(* Logix 5000 project; controller AdvManLab vendor 1 type 14 code 158 rev 28.12; software revision 28.01; part 6 of 13 *)
(* tags used below, declared in another part *)
   Out : P_PF52x_Out;   // Common part of PF523 / PF525 Output Assembly
   Inp_FwdPermOK : BOOL;   // 1=Permissives OK, drive can start Forward
   Inp_FwdNBPermOK : BOOL;   // 1=Non-Bypassable Permissives OK, drive can start Forward
   Inp_RevPermOK : BOOL;   // 1=Permissives OK, drive can start Reverse
   Inp_RevNBPermOK : BOOL;   // 1=Non-Bypassable Permissives OK, motor can start Reverse
   Inp_IntlkOK : BOOL;   // 1=Interlocks OK, drive can start/run
   Inp_NBIntlkOK : BOOL;   // 1=Non-Bypassable Interlocks OK, drive can start/run
   Inp_OvrdCmd : SINT;   // Override Mode Command: 0=None, 1=Stop, 2=Start Fwd 3=Start Rev
   Cfg_SetTrack : BOOL;   // 1=PSets track OSets in Oper, OSets track PSets in Prog, 0=no tracking
   Cfg_PCmdClear : ALIAS FOR Mode.Cfg_PCmdClear;
   Cfg_ShedOnFailToStart : BOOL;   // 1=Stop Motor and Alarm on Fail to Start; 0=Alarm only on Fail to Start
   Cfg_ShedOnIOFault : BOOL;   // 1=Stop Motor and Alarm on I/O Fault; 0=Alarm only on I/O Fault
   Cfg_FailToStartAckReqd : ALIAS FOR FailToStart.Cfg_AckReqd;   // 1=Acknowledge required for Fail to Start Alarm
   Cfg_FailToStopAckReqd : ALIAS FOR FailToStop.Cfg_AckReqd;   // 1=Acknowledge required for Fail to Stop Alarm
   Cfg_IntlkTripAckReqd : ALIAS FOR IntlkTrip.Cfg_AckReqd;   // 1=Acknowledge required for Interlock Trip Alarm
   Cfg_DriveFaultAckReqd : ALIAS FOR DriveFault.Cfg_AckReqd;   // 1=Acknowledge required for Drive Fault Alarm
   Cfg_IOFaultAckReqd : ALIAS FOR IOFault.Cfg_AckReqd;   // 1=Acknowledge required for I/O Fault Alarm
   Cfg_FailToStartSeverity : ALIAS FOR FailToStart.Cfg_Severity;   // Fail To Start Alarm Severity: 1..250=Low, 251..500=Medium, 501..750=High, 751..1000=Urgent
   Cfg_FailToStopSeverity : ALIAS FOR FailToStop.Cfg_Severity;   // Fail To Stop Alarm Severity: 1..250=Low, 251..500=Medium, 501..750=High, 751..1000=Urgent
   Cfg_IntlkTripSeverity : ALIAS FOR IntlkTrip.Cfg_Severity;   // Interlock Trip Alarm Severity: 1..250=Low, 251..500=Medium, 501..750=High, 751..1000=Urgent
   Cfg_DriveFaultSeverity : ALIAS FOR DriveFault.Cfg_Severity;   // Drive Fault Alarm Severity: 1..250=Low, 251..500=Medium, 501..750=High, 751..1000=Urgent
   Cfg_IOFaultSeverity : ALIAS FOR IOFault.Cfg_Severity;   // I/O Fault Alarm Severity: 1..250=Low, 251..500=Medium, 501..750=High, 751..1000=Urgent
   Cfg_MaxSpdRef : REAL;   // Maximum Speed Reference in EU (for limiting)
   Cfg_SpeedRefRawMax : INT;   // Speed Reference Maximum in Drive (raw) Units (for scaling)
   Cfg_SpeedRefEUMax : REAL;   // Speed Reference Maximum in Engineering Units (for scaling)
   Cfg_SpeedFdbkRawMax : INT;   // Speed Feedback Maximum in Drive (raw) Units (for scaling)
   Cfg_SpeedFdbkEUMax : REAL;   // Speed Feedback Maximum in Engineering Units (for scaling)
   Cfg_SimRampT : DINT;   // Time to ramp speed fdbk when in Simulation (sec)
   Cfg_FailToStartT : DINT;   // Time after Start to get Run Feedback before Fault (sec)
   Cfg_FailToStopT : DINT;   // Time after Stop to drop Run Feedback before Fault (sec)
   Cfg_ResetPulseT : DINT;   // Time to pulse Out_Reset to clear drive fault
   PSet_Owner : DINT;   // Program Owner Request ID (non-zero) or Release (zero)
   PCmd_Start : BOOL;   // Program Command to Start Drive
   PCmd_Stop : BOOL;   // Program Command to Stop Drive
   PCmd_Fwd : BOOL;   // Program Command to set direction to Fowrard
   PCmd_Rev : BOOL;   // Program Command to set direction to Reverse
   PCmd_Reset : BOOL;   // Program Command to Reset drive fault and all Alarms requiring Reset
   OCmd_Start : BOOL;   // Operator Command to Start Drive
   OCmd_Stop : BOOL;   // Operator Command to Stop Drive
   OCmd_Jog : BOOL;   // Operator Command to Jog Drive (not cleared by P_PF52x!)
   OCmd_Fwd : BOOL;   // Operator Command to set direction to Forward
   OCmd_Rev : BOOL;   // Operator Command to set direction to Reverse
   OCmd_Bypass : BOOL;   // Operator Command to Bypass all Bypassable Interlocks and Permissives
   OCmd_Check : BOOL;   // Operator Command to Check (not bypass) all Interlocks and Permissives
   MCmd_Disable : BOOL;   // Maintenance Command to Disable Drive
   MCmd_Enable : BOOL;   // Maintenance Command to Enable (allow to run) Drive
   OCmd_Reset : BOOL;   // Operator Command to Reset all Alarms requiring Reset
   OCmd_ResetAckAll : BOOL;   // Operator Command to Reset all Alarms and latched Shed conditions
   Val_SpeedRefEUMax : REAL;   // Maximum of Speed Reference = MAX (Cfg_SpeedFdbkEUMin, Cfg_SpeedFdbkEUMax)
   Val_SpeedFdbkEUMax : REAL;   // Maximum of Speed Feedback = MAX (Cfg_SpeedFdbkEUMin, Cfg_SpeedFdbkEUMax)
   Val_OutPower : REAL;   // Drive output power (kW)
   Val_Cmd : SINT;   // Device Command 0=None, 1=Stop, 2=StartFwd 3=StartRev 4=JogFwd 5=JogRev
   Val_Fdbk : SINT;   // Device Feedback 0=Stopped, 1=Running Fwd 2=Running Rev 3=Accelerating 4=Decelerating
   Val_Sts : SINT;   // Device Confirmed Sts 0? 1=Stop 2=RunF 3=RunR 4=JogF 5=JogR 6=Stopping 7=Starting F 8=Starting R, 33=Disabled
   Val_Fault : SINT;   // Device Fault Status 0=None, 16=Fail to Start, 17 = Fail to Stop, 18=Drive Fault, 32=I/O Fault, 34=Config Error
   Val_Mode : ALIAS FOR Mode.Val;
   Val_Owner : DINT;   // Current Object Owner ID (0=not owned)
   Sts_ActualDir : BOOL;   // 1=Drive Actual direction is Forward, 0=Reverse
   Nrdy_OperPrio : BOOL;   // 1=Device Not Ready: Operator State 0 Priority Command Requires Reset
   Nrdy_Fail : BOOL;   // 1=Device Not Ready: Device Failure (Shed Requires Reset)
   Nrdy_IOFault : BOOL;   // 1=Device Not Ready: I/O Fault (Shed Requires Reset)
   Ack_FailToStart : ALIAS FOR FailToStart.Ack;   // 1=Fail to Start Alarm has been acknowledged
   Ack_FailToStop : ALIAS FOR FailToStop.Ack;   // 1=Fail to Stop Alarm has been acknowledged
   Ack_IntlkTrip : ALIAS FOR IntlkTrip.Ack;   // 1=Interlock Trip Alarm has been acknowledged
   Ack_DriveFault : ALIAS FOR DriveFault.Ack;   // 1=Drive Fault Alarm has been acknowledged
   Ack_IOFault : ALIAS FOR IOFault.Ack;   // 1=I/O Fault Alarm has been acknowledged
   P_PF52x : BOOL;   // Unique Parameter Name for auto - discovery
   Mode : P_Mode;   // Drive Mode Selection
   Wrk_Run : BOOL;   // 1=Drive should be "running", 0=should be "stopped"
   Wrk_Jog : BOOL;   // 1=Jog Drive, 0=Drive not jogging
(* P_PF52x, continued *)

ROUTINE Prescan   (* ladder *)
// Clear Ownership, set drive to STOP, clear "lurking" Commands
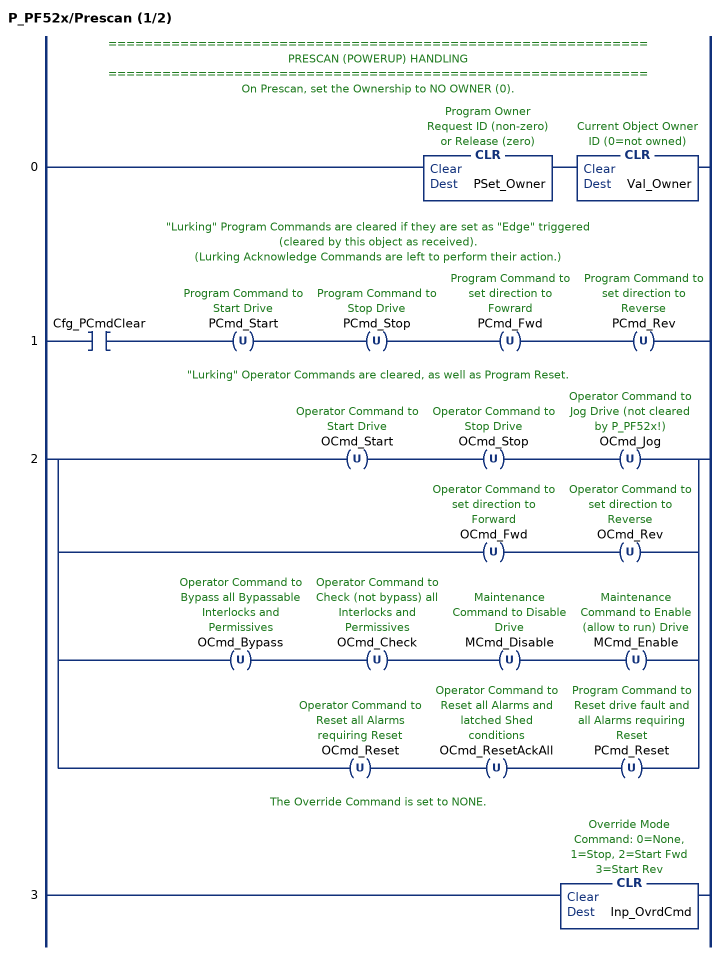
   // ============================================================
   // PRESCAN (POWERUP) HANDLING
   // ============================================================
   // On Prescan, set the Ownership to NO OWNER (0).
   0: CLR(PSet_Owner)CLR(Val_Owner);
   // "Lurking" Program Commands are cleared if they are set as "Edge" triggered
   // (cleared by this object as received).
   // (Lurking Acknowledge Commands are left to perform their action.)
   1: XIC(Cfg_PCmdClear)OTU(PCmd_Start)OTU(PCmd_Stop)OTU(PCmd_Fwd)OTU(PCmd_Rev);
   // "Lurking" Operator Commands are cleared, as well as Program Reset.
   2: [OTU(OCmd_Start) OTU(OCmd_Stop) OTU(OCmd_Jog) ,OTU(OCmd_Fwd) OTU(OCmd_Rev) ,OTU(OCmd_Bypass) OTU(OCmd_Check) OTU(MCmd_Disable) OTU(MCmd_Enable) ,OTU(OCmd_Reset) OTU(OCmd_ResetAckAll) OTU(PCmd_Reset) ];
   // The Override Command is set to NONE.
   3: CLR(Inp_OvrdCmd);
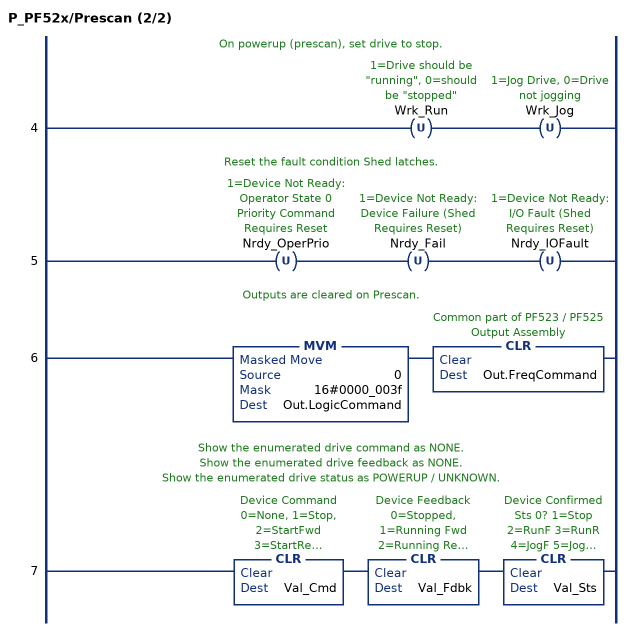
   // On powerup (prescan), set drive to stop.
   4: OTU(Wrk_Run)OTU(Wrk_Jog);
   // Reset the fault condition Shed latches.
   5: OTU(Nrdy_OperPrio)OTU(Nrdy_Fail)OTU(Nrdy_IOFault);
   // Outputs are cleared on Prescan.
   6: MVM(0,16#0000_003f,Out.LogicCommand)CLR(Out.FreqCommand);
   // Show the enumerated drive command as NONE.
   // Show the enumerated drive feedback as NONE.
   // Show the enumerated drive status as POWERUP / UNKNOWN.
   7: CLR(Val_Cmd)CLR(Val_Fdbk)CLR(Val_Sts);
END_ROUTINE
END_ADD_ON_INSTRUCTION

ADD_ON_INSTRUCTION PF525_Faceplate_AOI   (* revision 1.0 *)
// PF525 Drive FTView ME Faceplate AOI
VAR_INPUT
   Inp_NumRowsVis : DINT := 9;
   Set_FaceplateAnimation : INT;
END_VAR
VAR_OUTPUT
   Sts_ProgramModeEnabled : BOOL; {access Read Only}
   Sts_OperatorModeEnabled : BOOL; {access Read Only}
   Sts_DriveStatus_Faulted : BOOL; {access Read Only}
   Sts_DriveStatus_Active : BOOL; {access Read Only}
   Sts_DriveStatus_Ready : BOOL; {access Read Only}
   Sts_DriveStatus_Alarm : BOOL; {access Read Only}
   Sts_DriveStatus_AtSpeed : BOOL; {access Read Only}
   Sts_CommFault : BOOL; {access Read Only}
   Sts_DriveStatus_ActualDir : BOOL; {access Read Only}
   Sts_DeviceState : DINT; {access Read Only}
   Sts_Value1 : REAL; {access Read Only}
   Sts_Value2 : REAL; {access Read Only}
   Sts_Value3 : REAL; {access Read Only}
   Sts_Value4 : REAL; {access Read Only}
END_VAR
VAR_INPUT
   Set_TrendNextPenOper : DINT;
   Set_Value1Min : DINT;
   Set_Value1Max : DINT := 60;
   Set_Value2Min : DINT;
   Set_Value2Max : DINT := 1;
   Set_Value3Max : DINT := 1;
   Set_Value3Min : DINT;
END_VAR
VAR_OUTPUT
   Val_TrendMax : DINT; {access Read Only}
   Val_TrendMin : DINT; {access Read Only}
   Val_SpdFdbk_Units : DINT; {access Read Only}
   Val_Fault1Code : DINT; {access Read Only}
END_VAR
VAR_INPUT
   Cmd_OperOperReq : BOOL;
   Cmd_ProgOperReq : BOOL;
   Cmd_OperProgReq : BOOL;
   Cmd_ProgProgReq : BOOL;
   Cmd_StartOper : BOOL;
   Cmd_StartProg : BOOL;
   Cmd_StopOper : BOOL;
   Cmd_StopProg : BOOL;
   Cmd_ResetOper : BOOL;
   Cmd_ResetProg : BOOL;
   Cmd_JogOper : BOOL;
   Cmd_JogProg : BOOL;
   Cmd_FwdOper : BOOL;
   Cmd_FwdProg : BOOL;
   Cmd_RevOper : BOOL;
   Cmd_RevProg : BOOL;
   Cmd_OperToProgPermissive : BOOL := 1;
   Cmd_ProgToOperPermissive : BOOL := 1;
   Set_SpeedOper : INT;
END_VAR
VAR_IN_OUT
   Inp_PowerFlex_525 : AB:PowerFlex525V_E_8A02D441:I:0; {required}
   Out_PowerFlex_525 : AB:PowerFlex525V_E_5483BAFD:O:0; {required}
END_VAR
VAR_INPUT
   Cmd_MOPIncProg : BOOL;
   Cmd_MOPIncOper : BOOL;
   Cmd_Accel1Oper : BOOL;
   Cmd_Accel2Oper : BOOL;
   Cmd_Decel1Oper : BOOL;
   Cmd_Decel2Oper : BOOL;
   Cmd_Accel1Prog : BOOL;
   Cmd_Accel2Prog : BOOL;
   Cmd_Decel1Prog : BOOL;
   Cmd_Decel2Prog : BOOL;
   Cmd_MOPDecProg : BOOL;
   Cmd_MOPDecOper : BOOL;
   Set_AccelProg : REAL;
   Set_DecelProg : REAL;
   Set_CommFaultTimerPresetProg : DINT := 10000;
   Cmd_LocalContrlProg : BOOL;
   Cmd_LocalContrlOper : BOOL;
   Cmd_FreqSel01Prog : BOOL;
   Cmd_FreqSel01Oper : BOOL;
   Cmd_FreqSel02Prog : BOOL;
   Cmd_FreqSel02Oper : BOOL;
   Cmd_FreqSel03Prog : BOOL;
   Cmd_FreqSel03Oper : BOOL;
   Set_SpeedProg : INT;
   Set_CommFaultTimerPresetOper : DINT;
   Set_DecelOper : REAL;
   Set_AccelOper : REAL;
   Inp_FaultCode : DINT;   // Fault Code
   NotReady_Fault : BOOL;
   CLEAR_Fault : BOOL;
   Module_FaultTrigger : BOOL;
   Module_FaultCode : DINT;
   RESET_Fault : BOOL;
   Inp_Display_Val_1 : REAL;
   Inp_Display_Val_2 : REAL;
   Inp_Display_Val_3 : REAL;
   Inp_Display_Val_4 : REAL;
   Comm_Status : DINT;
   Sts_DriveStatus_CommFault : BOOL;
   Inst_Error : BOOL;
END_VAR
VAR_IN_OUT
   LastFault_Msg : MESSAGE; {required}
END_VAR
VAR_INPUT
   LastFaultCode : DINT;
   SpdRef_Units : INT;
   SpdScaler60Hz : REAL; {required}
   GearRatio : REAL; {required}
   Out_SpdRef_Units : DINT;
   Val_OutputFreq : REAL;
   Val_OutputCurrent : REAL;
   Val_OutputVoltage : DINT;
END_VAR
VAR_OUTPUT
   Sts_PowerflexAlarmTrigger : DINT; {access Read Only}
   Controller_trigger : BOOL; {access Read Only}
END_VAR
VAR
   Set_Value4Units : STRING := 'units';
   Set_Value3Units : STRING := 'units';
   Set_Value2Units : STRING := 'Amps';
   Set_Value1Units : STRING := 'Hz';
   Set_SpeedUnitsOper : STRING := 'Hz';
   Set_DeviceNameOper : STRING := 'PF525';
   Set_Value3Name : STRING := 'Value 3';
   Set_Value2Name : STRING := 'curr fdbk';
   Set_Value1Name : STRING := 'unit fdbk';
   Set_Value4Name : STRING := 'Value 4';
   OperONS : BOOL; {access None}
   CommFaultTimer : TIMER := (PRE := 10000); {access None}
   Trigger_ONS : BOOL;
   Trigger_Delay_Timer : TIMER; {access None}
   Handshake_Initial_Status : BOOL;
   Comm_Loss_Delay_Timer : TIMER; {access None}
   storage_bit2 : BOOL; {access None}
END_VAR

ROUTINE Logic   (* ladder *)
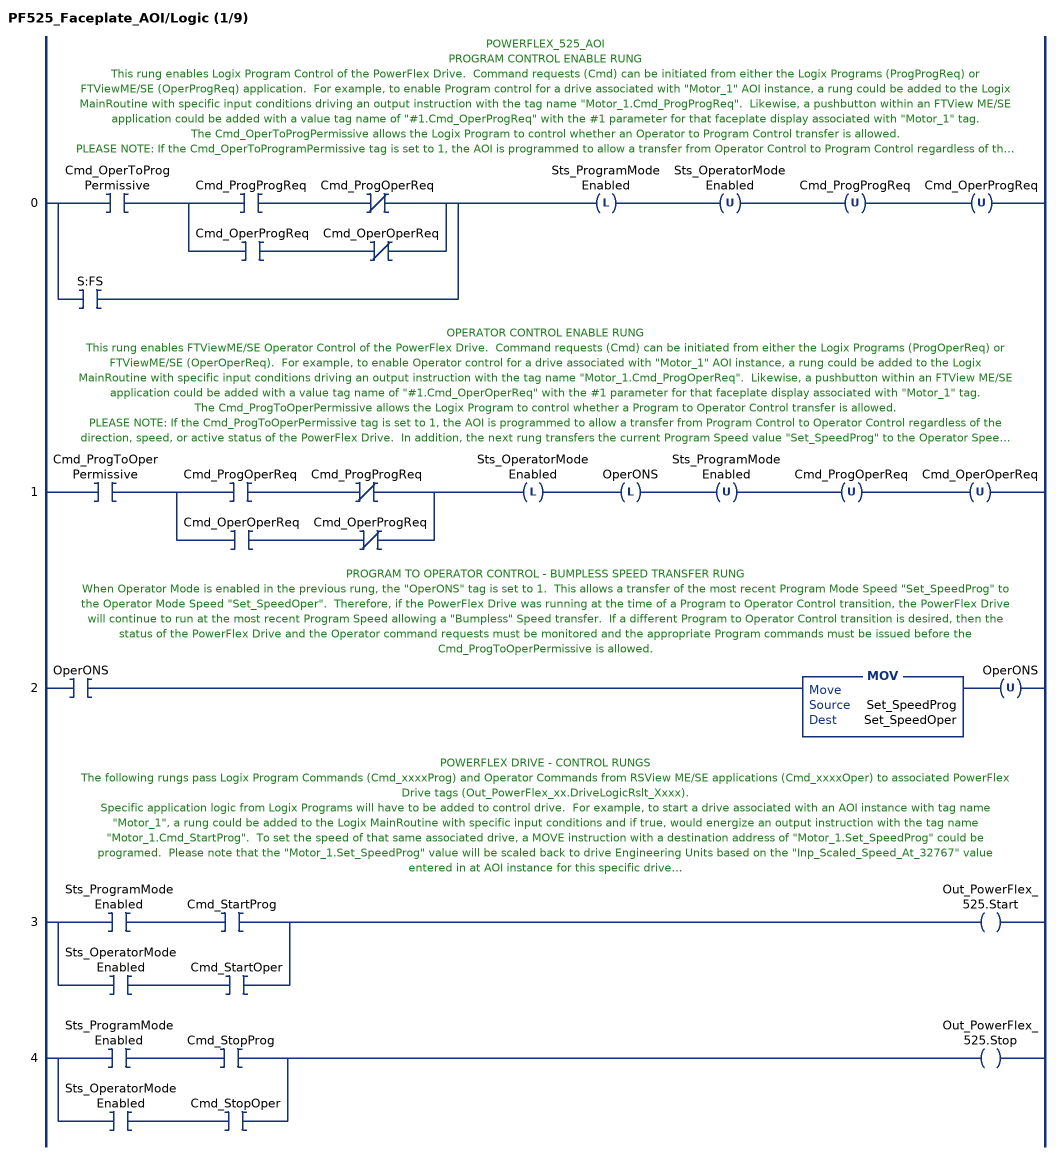
   // POWERFLEX_525_AOI
   // PROGRAM CONTROL ENABLE RUNG
   // This rung enables Logix Program Control of the PowerFlex Drive.  Command requests (Cmd) can be initiated from either the Logix Programs (ProgProgReq) or FTViewME/SE (OperProgReq) application.  For example, to enable Program control for a drive associated with "Motor_1" AOI instance, a rung could be added to the Logix MainRoutine with specific input conditions driving an output instruction with the tag name "Motor_1.Cmd_ProgProgReq".  Likewise, a pushbutton within an FTView ME/SE application could be added with a value tag name of "#1.Cmd_OperProgReq" with the #1 parameter for that faceplate display associated with "Motor_1" tag.
   // The Cmd_OperToProgPermissive allows the Logix Program to control whether an Operator to Program Control transfer is allowed.
   // PLEASE NOTE: If the Cmd_OperToProgramPermissive tag is set to 1, the AOI is programmed to allow a transfer from Operator Control to Program Control regardless of the direction, speed, or active status of the PowerFlex Drive.  Therefore, the status of the PowerFlex Drive must be monitored and used to set Cmd_OperToProgramPermissive tag outside of the AOI to insure a safe transfer.
   0: [XIC(Cmd_OperToProgPermissive) [XIC(Cmd_ProgProgReq) XIO(Cmd_ProgOperReq) ,XIC(Cmd_OperProgReq) XIO(Cmd_OperOperReq) ] ,XIC(S:FS) ]OTL(Sts_ProgramModeEnabled)OTU(Sts_OperatorModeEnabled)OTU(Cmd_ProgProgReq)OTU(Cmd_OperProgReq);
   // OPERATOR CONTROL ENABLE RUNG
   // This rung enables FTViewME/SE Operator Control of the PowerFlex Drive.  Command requests (Cmd) can be initiated from either the Logix Programs (ProgOperReq) or FTViewME/SE (OperOperReq).  For example, to enable Operator control for a drive associated with "Motor_1" AOI instance, a rung could be added to the Logix MainRoutine with specific input conditions driving an output instruction with the tag name "Motor_1.Cmd_ProgOperReq".  Likewise, a pushbutton within an FTView ME/SE application could be added with a value tag name of "#1.Cmd_OperOperReq" with the #1 parameter for that faceplate display associated with "Motor_1" tag.
   // The Cmd_ProgToOperPermissive allows the Logix Program to control whether a Program to Operator Control transfer is allowed.
   // PLEASE NOTE: If the Cmd_ProgToOperPermissive tag is set to 1, the AOI is programmed to allow a transfer from Program Control to Operator Control regardless of the direction, speed, or active status of the PowerFlex Drive.  In addition, the next rung transfers the current Program Speed value "Set_SpeedProg" to the Operator Speed tag, "Set_SpeedOper" tag, creating a "bumpless" transfer when a transfer from Program Control to Operator Control is executed.  Therefore, the status of the PowerFlex Drive must be monitored and appropriate Program commands, for the specific application, must be issued before the Cmd_ProgToOperPermissive tag is set, to insure a safe Program to Operator Control transfer.
   1: XIC(Cmd_ProgToOperPermissive)[XIC(Cmd_ProgOperReq) XIO(Cmd_ProgProgReq) ,XIC(Cmd_OperOperReq) XIO(Cmd_OperProgReq) ]OTL(Sts_OperatorModeEnabled)OTL(OperONS)OTU(Sts_ProgramModeEnabled)OTU(Cmd_ProgOperReq)OTU(Cmd_OperOperReq);
   // PROGRAM TO OPERATOR CONTROL - BUMPLESS SPEED TRANSFER RUNG
   // When Operator Mode is enabled in the previous rung, the "OperONS" tag is set to 1.  This allows a transfer of the most recent Program Mode Speed "Set_SpeedProg" to the Operator Mode Speed "Set_SpeedOper".  Therefore, if the PowerFlex Drive was running at the time of a Program to Operator Control transition, the PowerFlex Drive will continue to run at the most recent Program Speed allowing a "Bumpless" Speed transfer.  If a different Program to Operator Control transition is desired, then the status of the PowerFlex Drive and the Operator command requests must be monitored and the appropriate Program commands must be issued before the Cmd_ProgToOperPermissive is allowed.
   2: XIC(OperONS)MOV(Set_SpeedProg,Set_SpeedOper)OTU(OperONS);
   // POWERFLEX DRIVE - CONTROL RUNGS
   // The following rungs pass Logix Program Commands (Cmd_xxxxProg) and Operator Commands from RSView ME/SE applications (Cmd_xxxxOper) to associated PowerFlex Drive tags (Out_PowerFlex_xx.DriveLogicRslt_Xxxx).
   // Specific application logic from Logix Programs will have to be added to control drive.  For example, to start a drive associated with an AOI instance with tag name "Motor_1", a rung could be added to the Logix MainRoutine with specific input conditions and if true, would energize an output instruction with the tag name "Motor_1.Cmd_StartProg".  To set the speed of that same associated drive, a MOVE instruction with a destination address of "Motor_1.Set_SpeedProg" could be programed.  Please note that the "Motor_1.Set_SpeedProg" value will be scaled back to drive Engineering Units based on the "Inp_Scaled_Speed_At_32767" value entered in at AOI instance for this specific drive.
   // Commands from FTView ME/SE applications will also control the drive when Operator Mode is enabled.  For example, to start a drive associated with "Motor_1" AOI instance, a pushbutton within an FTView ME application with a tag name of "#1.Cmd_StartOper" would have to be configured.  The #1 parameter tagname for that faceplate display would have to be "Motor_1".  To set the speed of that same "Motor_1" associated drive, a numeric input object with the tag name of "#1.Set_SpeedOper" would have to be configured.  Please note that the "#1.Set_SpeedOper" value will be scaled back to drive Engineering Units based on the "Inp_Scaled_Speed_At_32767" value entered in at AOI instance for this specific drive.
   // For ability to set AccelTime1 and DecelTime1, the datalinks within the PowerFlex Drive Module Definitions need to be assigned to these drive parameters.
   3: [XIC(Sts_ProgramModeEnabled) XIC(Cmd_StartProg) ,XIC(Sts_OperatorModeEnabled) XIC(Cmd_StartOper) ]OTE(Out_PowerFlex_525.Start);
   4: [XIC(Sts_ProgramModeEnabled) XIC(Cmd_StopProg) ,XIC(Sts_OperatorModeEnabled) XIC(Cmd_StopOper) ]OTE(Out_PowerFlex_525.Stop);
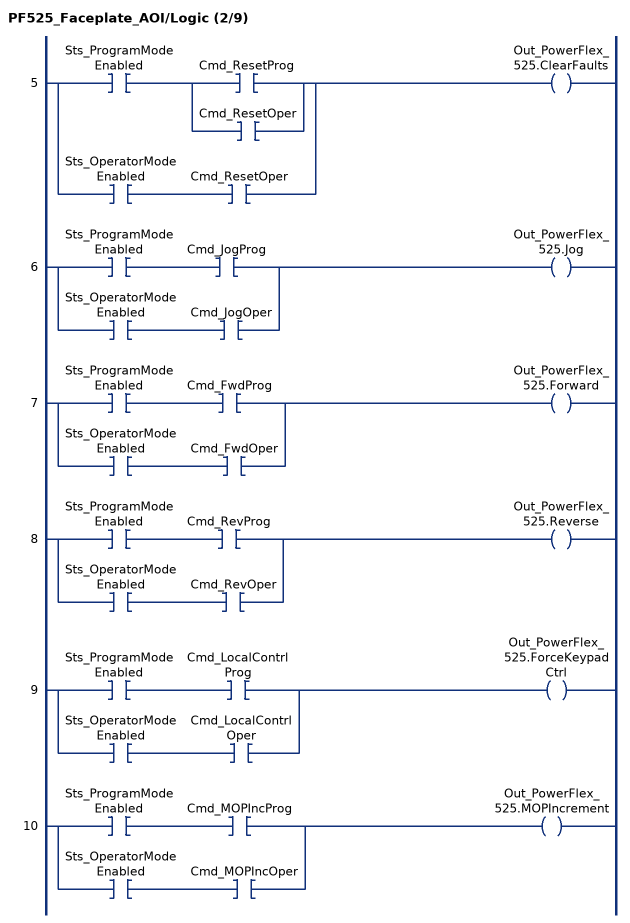
   5: [XIC(Sts_ProgramModeEnabled) [XIC(Cmd_ResetProg) ,XIC(Cmd_ResetOper) ] ,XIC(Sts_OperatorModeEnabled) XIC(Cmd_ResetOper) ]OTE(Out_PowerFlex_525.ClearFaults);
   6: [XIC(Sts_ProgramModeEnabled) XIC(Cmd_JogProg) ,XIC(Sts_OperatorModeEnabled) XIC(Cmd_JogOper) ]OTE(Out_PowerFlex_525.Jog);
   7: [XIC(Sts_ProgramModeEnabled) XIC(Cmd_FwdProg) ,XIC(Sts_OperatorModeEnabled) XIC(Cmd_FwdOper) ]OTE(Out_PowerFlex_525.Forward);
   8: [XIC(Sts_ProgramModeEnabled) XIC(Cmd_RevProg) ,XIC(Sts_OperatorModeEnabled) XIC(Cmd_RevOper) ]OTE(Out_PowerFlex_525.Reverse);
   9: [XIC(Sts_ProgramModeEnabled) XIC(Cmd_LocalContrlProg) ,XIC(Sts_OperatorModeEnabled) XIC(Cmd_LocalContrlOper) ]OTE(Out_PowerFlex_525.ForceKeypadCtrl);
   10: [XIC(Sts_ProgramModeEnabled) XIC(Cmd_MOPIncProg) ,XIC(Sts_OperatorModeEnabled) XIC(Cmd_MOPIncOper) ]OTE(Out_PowerFlex_525.MOPIncrement);
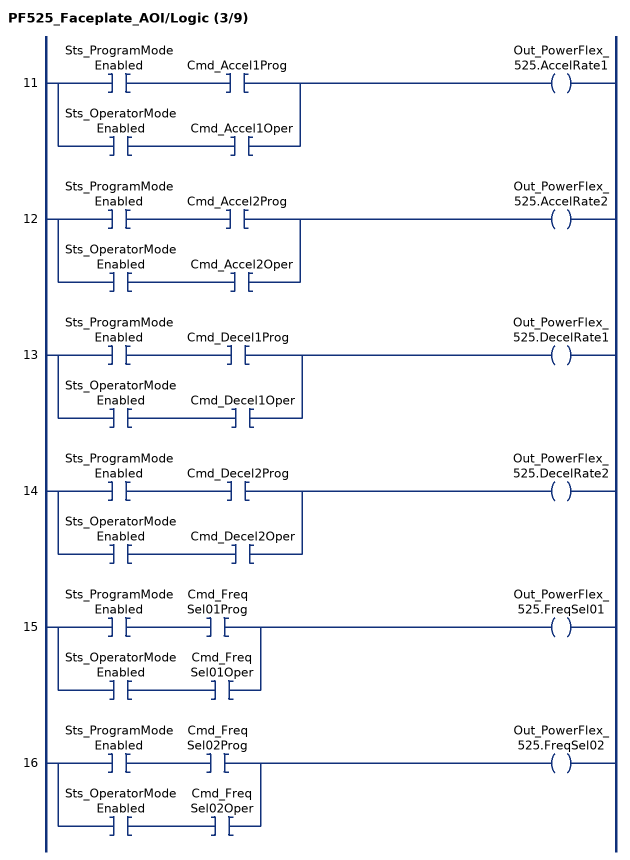
   11: [XIC(Sts_ProgramModeEnabled) XIC(Cmd_Accel1Prog) ,XIC(Sts_OperatorModeEnabled) XIC(Cmd_Accel1Oper) ]OTE(Out_PowerFlex_525.AccelRate1);
   12: [XIC(Sts_ProgramModeEnabled) XIC(Cmd_Accel2Prog) ,XIC(Sts_OperatorModeEnabled) XIC(Cmd_Accel2Oper) ]OTE(Out_PowerFlex_525.AccelRate2);
   13: [XIC(Sts_ProgramModeEnabled) XIC(Cmd_Decel1Prog) ,XIC(Sts_OperatorModeEnabled) XIC(Cmd_Decel1Oper) ]OTE(Out_PowerFlex_525.DecelRate1);
   14: [XIC(Sts_ProgramModeEnabled) XIC(Cmd_Decel2Prog) ,XIC(Sts_OperatorModeEnabled) XIC(Cmd_Decel2Oper) ]OTE(Out_PowerFlex_525.DecelRate2);
   15: [XIC(Sts_ProgramModeEnabled) XIC(Cmd_FreqSel01Prog) ,XIC(Sts_OperatorModeEnabled) XIC(Cmd_FreqSel01Oper) ]OTE(Out_PowerFlex_525.FreqSel01);
   16: [XIC(Sts_ProgramModeEnabled) XIC(Cmd_FreqSel02Prog) ,XIC(Sts_OperatorModeEnabled) XIC(Cmd_FreqSel02Oper) ]OTE(Out_PowerFlex_525.FreqSel02);
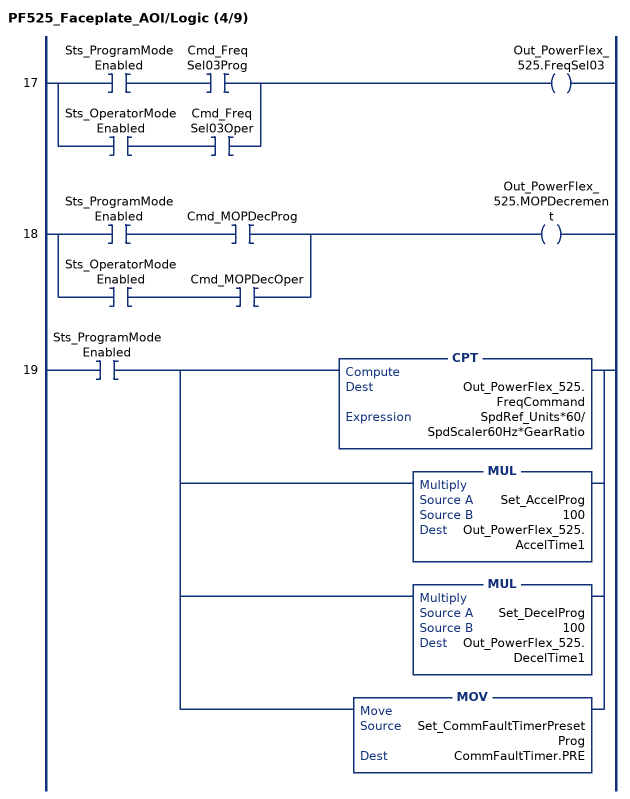
   17: [XIC(Sts_ProgramModeEnabled) XIC(Cmd_FreqSel03Prog) ,XIC(Sts_OperatorModeEnabled) XIC(Cmd_FreqSel03Oper) ]OTE(Out_PowerFlex_525.FreqSel03);
   18: [XIC(Sts_ProgramModeEnabled) XIC(Cmd_MOPDecProg) ,XIC(Sts_OperatorModeEnabled) XIC(Cmd_MOPDecOper) ]OTE(Out_PowerFlex_525.MOPDecrement);
   19: XIC(Sts_ProgramModeEnabled)[CPT(Out_PowerFlex_525.FreqCommand,SpdRef_Units*60/SpdScaler60Hz*GearRatio) ,MUL(Set_AccelProg,100,Out_PowerFlex_525.AccelTime1) ,MUL(Set_DecelProg,100,Out_PowerFlex_525.DecelTime1) ,MOV(Set_CommFaultTimerPresetProg,CommFaultTimer.PRE) ];
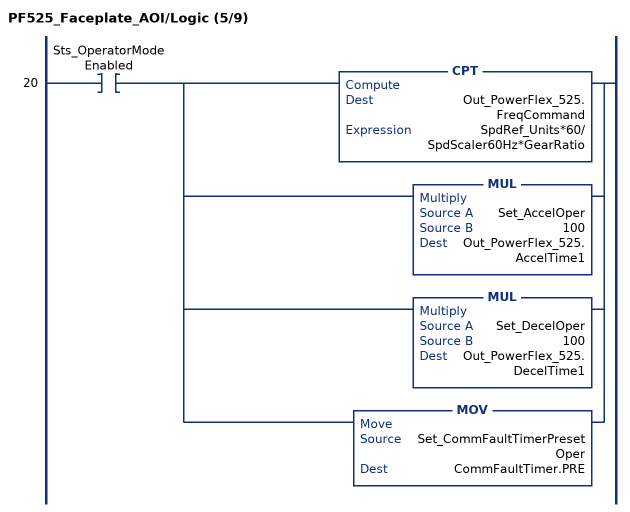
   20: XIC(Sts_OperatorModeEnabled)[CPT(Out_PowerFlex_525.FreqCommand,SpdRef_Units*60/SpdScaler60Hz*GearRatio) ,MUL(Set_AccelOper,100,Out_PowerFlex_525.AccelTime1) ,MUL(Set_DecelOper,100,Out_PowerFlex_525.DecelTime1) ,MOV(Set_CommFaultTimerPresetOper,CommFaultTimer.PRE) ];
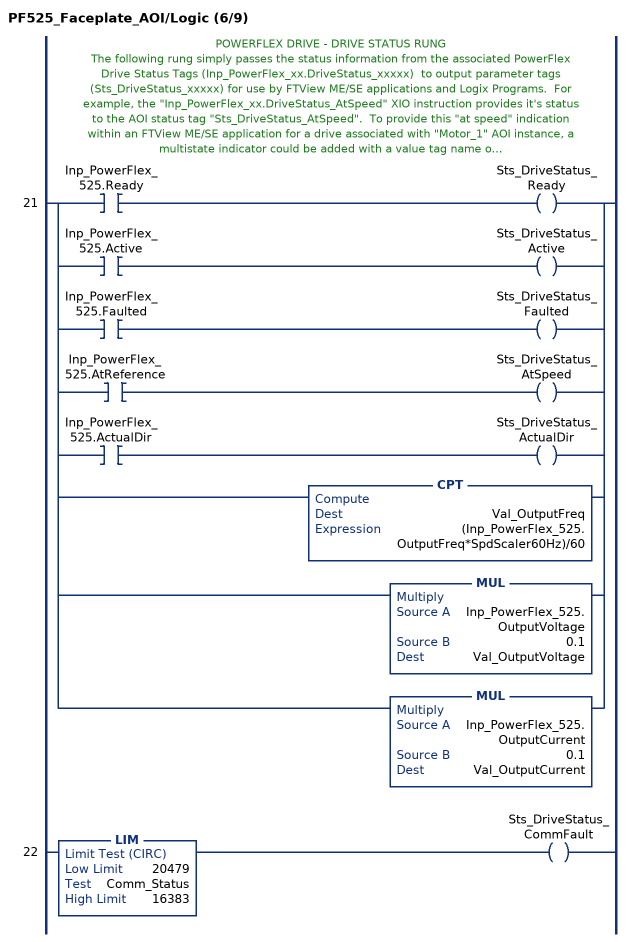
   // POWERFLEX DRIVE - DRIVE STATUS RUNG
   // The following rung simply passes the status information from the associated PowerFlex Drive Status Tags (Inp_PowerFlex_xx.DriveStatus_xxxxx)  to output parameter tags (Sts_DriveStatus_xxxxx) for use by FTView ME/SE applications and Logix Programs.  For example, the "Inp_PowerFlex_xx.DriveStatus_AtSpeed" XIO instruction provides it's status to the AOI status tag "Sts_DriveStatus_AtSpeed".  To provide this "at speed" indication within an FTView ME/SE application for a drive associated with "Motor_1" AOI instance, a multistate indicator could be added with a value tag name of "#1.Sts_DriveStatus_AtSpeed".  The #1 parameter for the faceplate display with the at speed indicator associated with "Motor_1" would be assigned the "Motor_1" tag.  To use this "Sts_DriveStatus_AtSpeed" status for the drive associated with "Motor_1" within a Logix Program routine you would simply assign an input instruction with a tag name of Motor_1.Sts_ DriveStatus_AtSpeed.  Please note that the "Val_OutputFreq" value used by the FTView ME/SE application is scaled based on the "Inp_Scaled_Speed_At_60Hz" value entered in at AOI instance for the specific drive.
   21: [XIC(Inp_PowerFlex_525.Ready) OTE(Sts_DriveStatus_Ready) ,XIC(Inp_PowerFlex_525.Active) OTE(Sts_DriveStatus_Active) ,XIC(Inp_PowerFlex_525.Faulted) OTE(Sts_DriveStatus_Faulted) ,XIC(Inp_PowerFlex_525.AtReference) OTE(Sts_DriveStatus_AtSpeed) ,XIC(Inp_PowerFlex_525.ActualDir) OTE(Sts_DriveStatus_ActualDir) ,CPT(Val_OutputFreq,(Inp_PowerFlex_525.OutputFreq*SpdScaler60Hz)/60) ,MUL(Inp_PowerFlex_525.OutputVoltage,0.1,Val_OutputVoltage) ,MUL(Inp_PowerFlex_525.OutputCurrent,0.1,Val_OutputCurrent) ];
   22: LIM(20479,Comm_Status,16383)OTE(Sts_DriveStatus_CommFault);
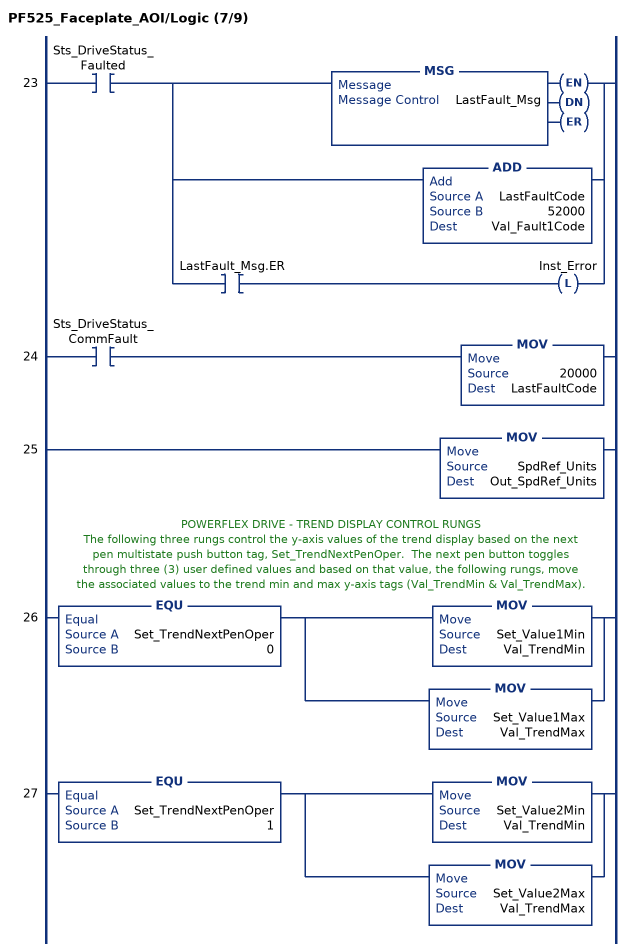
   23: XIC(Sts_DriveStatus_Faulted)[MSG(LastFault_Msg) ,ADD(LastFaultCode,52000,Val_Fault1Code) ,XIC(LastFault_Msg.ER) OTL(Inst_Error) ];
   24: XIC(Sts_DriveStatus_CommFault)MOV(20000,LastFaultCode);
   25: MOV(SpdRef_Units,Out_SpdRef_Units);
   // POWERFLEX DRIVE - TREND DISPLAY CONTROL RUNGS
   // The following three rungs control the y-axis values of the trend display based on the next pen multistate push button tag, Set_TrendNextPenOper.  The next pen button toggles through three (3) user defined values and based on that value, the following rungs, move the associated values to the trend min and max y-axis tags (Val_TrendMin & Val_TrendMax).
   26: EQU(Set_TrendNextPenOper,0)[MOV(Set_Value1Min,Val_TrendMin) ,MOV(Set_Value1Max,Val_TrendMax) ];
   27: EQU(Set_TrendNextPenOper,1)[MOV(Set_Value2Min,Val_TrendMin) ,MOV(Set_Value2Max,Val_TrendMax) ];
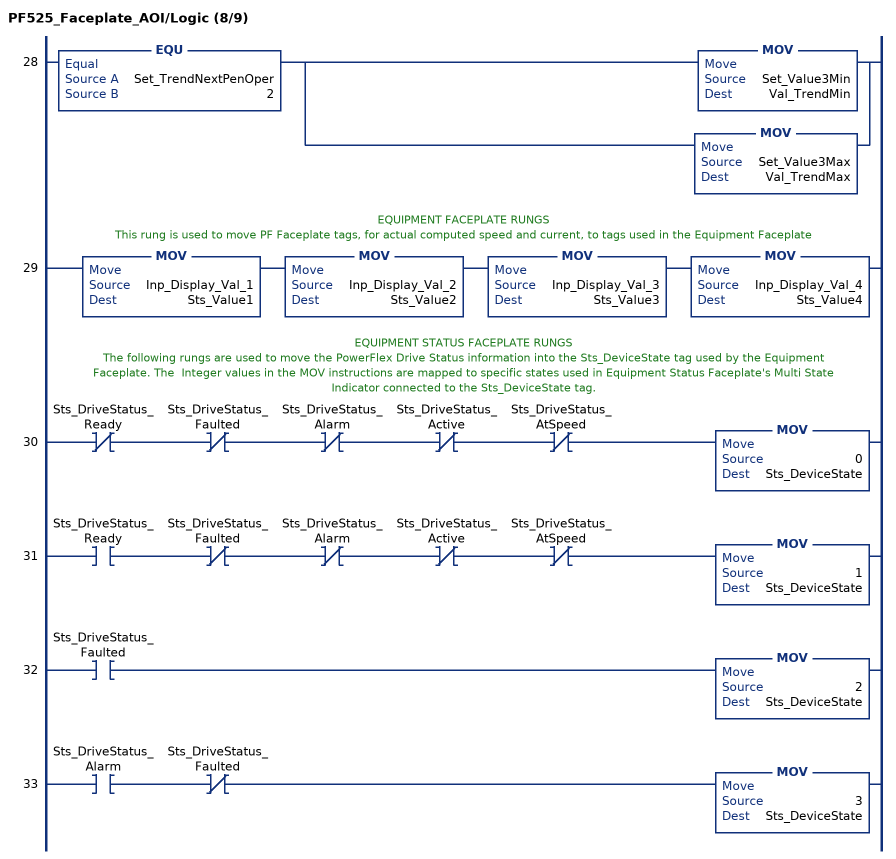
   28: EQU(Set_TrendNextPenOper,2)[MOV(Set_Value3Min,Val_TrendMin) ,MOV(Set_Value3Max,Val_TrendMax) ];
   // EQUIPMENT FACEPLATE RUNGS
   // This rung is used to move PF Faceplate tags, for actual computed speed and current, to tags used in the Equipment Faceplate
   29: MOV(Inp_Display_Val_1,Sts_Value1)MOV(Inp_Display_Val_2,Sts_Value2)MOV(Inp_Display_Val_3,Sts_Value3)MOV(Inp_Display_Val_4,Sts_Value4);
   // EQUIPMENT STATUS FACEPLATE RUNGS
   // The following rungs are used to move the PowerFlex Drive Status information into the Sts_DeviceState tag used by the Equipment Faceplate. The  Integer values in the MOV instructions are mapped to specific states used in Equipment Status Faceplate's Multi State Indicator connected to the Sts_DeviceState tag.
   30: XIO(Sts_DriveStatus_Ready)XIO(Sts_DriveStatus_Faulted)XIO(Sts_DriveStatus_Alarm)XIO(Sts_DriveStatus_Active)XIO(Sts_DriveStatus_AtSpeed)MOV(0,Sts_DeviceState);
   31: XIC(Sts_DriveStatus_Ready)XIO(Sts_DriveStatus_Faulted)XIO(Sts_DriveStatus_Alarm)XIO(Sts_DriveStatus_Active)XIO(Sts_DriveStatus_AtSpeed)MOV(1,Sts_DeviceState);
   32: XIC(Sts_DriveStatus_Faulted)MOV(2,Sts_DeviceState);
   33: XIC(Sts_DriveStatus_Alarm)XIO(Sts_DriveStatus_Faulted)MOV(3,Sts_DeviceState);
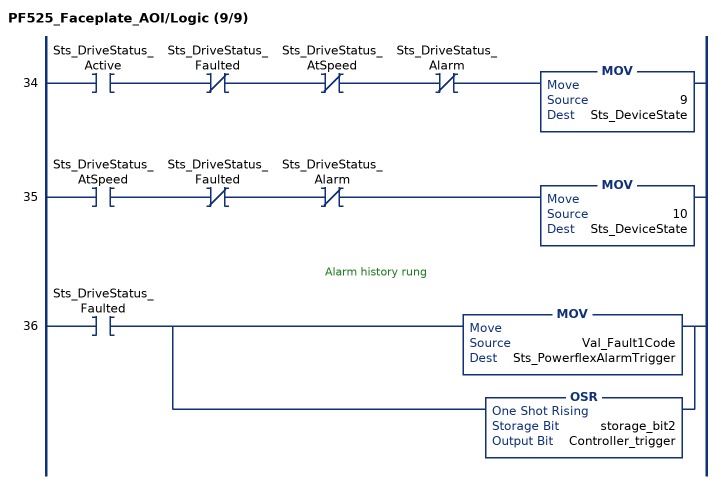
   34: XIC(Sts_DriveStatus_Active)XIO(Sts_DriveStatus_Faulted)XIO(Sts_DriveStatus_AtSpeed)XIO(Sts_DriveStatus_Alarm)MOV(9,Sts_DeviceState);
   35: XIC(Sts_DriveStatus_AtSpeed)XIO(Sts_DriveStatus_Faulted)XIO(Sts_DriveStatus_Alarm)MOV(10,Sts_DeviceState);
   // Alarm history rung
   36: XIC(Sts_DriveStatus_Faulted)[MOV(Val_Fault1Code,Sts_PowerflexAlarmTrigger) ,OSR(storage_bit2,Controller_trigger) ];
END_ROUTINE
END_ADD_ON_INSTRUCTION

VAR_GLOBAL   (* controller tags *)
   _SFS : MESSAGE;
   ABB_Loop_Conv_ES_Ch1 : BOOL := 1;   // Cell 3 Conveyor Pull Cord / E-Stop Ch1
   ABB_Loop_Conv_ES_Ch2 : BOOL := 1;   // Cell 3 Conveyor Pull Cord / E-Stop Ch2
   ABB_Loop_Conv_Safety_OK : BOOL := 1;
   ABB_Loop_Speed : DINT;
   ABBLoopPullCordES : EMERGENCY_STOP := (ChannelA := 1, ChannelB := 1, O1 := 1);   // EStop / Cable On ABB Loop
   ABBLoopPullCordESCH1 : BOOL;   // Cell 3 pull Cord CH1
   ABBLoopPullCordESCH2 : BOOL;   // Cell 3 pull Cord CH2
   ABBLoopSTO_O1 : BOOL := 1;
   ABBLoopSTO_O2 : BOOL := 1;
   ABBLoopVFD : PF525_Faceplate_AOI := (Inp_NumRowsVis := 9, Sts_ProgramModeEnabled := 1, Sts_DriveStatus_Faulted := 1, Sts_DriveStatus_ActualDir := 1, Sts_DeviceState := 2, Set_Value1Max := 60, Set_Value2Max := 1, Set_Value3Max := 1, Val_TrendMax := 60, Val_Fault1Code := 52105, Cmd_OperToProgPermissive := 1, Cmd_ProgToOperPermissive := 1, Set_CommFaultTimerPresetProg := 10000, Comm_Status := 16384, Inst_Error := 1, LastFaultCode := 105, SpdRef_Units := 30, SpdScaler60Hz := 1.0, GearRatio := 1.0, Out_SpdRef_Units := 30, Sts_PowerflexAlarmTrigger := 52105);
   Advance_Slide : BOOL := 1;
   AlwaysOff : BOOL;
   AlwaysOffSafe : BOOL;
   ASynch : BOOL;
   Auto_Valves01 : SINT := 85;
   Auto_Valves02 : SINT := 101;
   Auto_Valves_Safe01 : SINT := 85;
   Auto_Valves_Safe02 : SINT := 101;
   AutoDelay : TIMER := (PRE := 2000);
   AutoProgStart : TIMER := (PRE := 1000);
   AutoRun : BOOL;   // Run System in Automatic
   BobsBits : DINT := 65888;
        .0   // Test bit to trigger part to CNC3
   BobsTimer01 : TIMER := (PRE := 30000);   // Robot Drop Off simulation
   BobsTimer02 : TIMER := (PRE := 30000);
   C1_Robot_ES_OK : BOOL := 1;
   C1_Robot_Gates_OK : BOOL;
   C1EASRelay_Monitor : BOOL;   // Robot External Safety Gate Relay Monitor
   C1EESRelay_Monitor : BOOL;   // Robot External EStop Relay Monitor
   C1HoldBack : PalletStop := (Ext := 1);
   C1RobotStop : PalletStop := (Ext := 1);
   C1RobotStopPalletTransit : TIMER := (PRE := 500);
   C1RobotStopRetractConditions : BOOL;
   C1S : Fanuc_Cell_Safe := (CNC_A.LC_Ch1 := 1, CNC_A.LC_Ch2 := 1, CNC_A.EStop_Ch1 := 1, CNC_A.EStop_Ch2 := 1, CNC_B.LC_Ch1 := 1, CNC_B.LC_Ch2 := 1, CNC_B.DoorSW_Ch1 := 1, CNC_B.DoorSW_Ch2 := 1, CNC_B.EStop_Ch1 := 1, CNC_B.EStop_Ch2 := 1, Perim.GateSW_Ch1 := 1, Perim.GateSW_Ch2 := 1, Perim.Exit_LC_Ch1 := 1, Perim.Exit_LC_Ch2 := 1, Perim.Exit_Mute1 := 1, Perim.Exit_Mute2 := 1, Perim.EntMuteStatOK := 1, Perim.ExitMuteStatOK := 1, Perim.Exit_LC_Not_Blocked := 1); {produced}
        .CNC_A.LC_Ch2   // CNC1 Light Screen Ch2
        .CNC_A.DoorSW_Ch2   // CNC1 Door Switch Ch2
        .CNC_A.LC_Ch1   // CNC1 Light Screen Ch1
        .CNC_A.DoorSW_Ch1   // CNC1 Door Switch Ch1
        .CNC_B.LC_Ch2   // CNC2 Light Screen Ch2
        .CNC_B.DoorSW_Ch2   // CNC2 Door Switch Ch2
        .CNC_B.LC_Ch1   // CNC2 Light Screen Ch1
        .CNC_B.DoorSW_Ch1   // CNC2 Door Switch Ch1
        .Perim.GateSW_Ch1   // Cell 1 Gate Switch Ch1
        .Perim.GateSW_Ch2   // Cell 1 Gate Switch Ch2
        .Perim.Ent_LC_Ch1   // Cell 1 Entry Light Screen Ch1
        .Perim.Ent_LC_Ch2   // Cell 1 Entry Light Screen Ch2
        .Perim.Exit_LC_Ch1   // Cell 1 Exit Light Screen Ch1
        .Perim.Exit_LC_Ch2   // Cell 1 Exit Light Screen Ch2
        .Perim.Ent_Mute1   // Entry Mute 1 (Mute Signals Inverted)
        .Perim.Ent_Mute2   // Entry Mute 2 (Mute Signals Inverted)
        .Perim.Exit_Mute1   // Exit Mute 1 (Mute Signals Inverted)
        .Perim.Exit_Mute2   // Exit Mute 2 (Mute Signals Inverted)
   C21PartInTransit : TIMER := (PRE := 8000);
   C23Diverter : PalletStop := (Ext := 1);
   C23DivHoldBack : PalletStop := (Ext := 1);
   C23DivHoldBackRetractConditions : BOOL;
   C23DivHoldBackTransit : TIMER := (PRE := 500);
   C23PartInTransit : TIMER := (PRE := 11000);
   C2_Robot_ES_OK : BOOL := 1;
   C2_Robot_Gates_OK : BOOL := 1;
   C2EASRelay_Monitor : BOOL;   // Robot External Safety Gate Relay Monitor
   C2EESRelay_Monitor : BOOL;   // Robot External EStop Relay Monitor
   C2HoldBack : PalletStop := (Ext := 1);
   C2RobotStop : PalletStop := (Ext := 1);
   C2RobotStopPalletTransit : TIMER := (PRE := 500);
   C2RobotStopRetractConditions : BOOL;
   C2S : Fanuc_Cell_Safe := (CNC_A.LC_Ch1 := 1, CNC_A.LC_Ch2 := 1, CNC_B.LC_Ch1 := 1, CNC_B.LC_Ch2 := 1, CNC_B.EStop_Ch1 := 1, CNC_B.EStop_Ch2 := 1, Perim.GateSW_Ch1 := 1, Perim.GateSW_Ch2 := 1, Perim.Ent_LC_Ch1 := 1, Perim.Ent_LC_Ch2 := 1, Perim.Exit_LC_Ch1 := 1, Perim.Exit_LC_Ch2 := 1, Perim.Ent_Mute1 := 1, Perim.Ent_Mute2 := 1, Perim.Exit_Mute1 := 1, Perim.Exit_Mute2 := 1, Perim.EntMuteStatOK := 1, Perim.ExitMuteStatOK := 1, Perim.OK := 1, Perim.Ent_LC_Not_Blocked := 1, Perim.Exit_LC_Not_Blocked := 1); {produced}
        .CNC_A.LC_Ch2   // CNC3 Light Screen Ch2
        .CNC_A.DoorSW_Ch2   // CNC3 Door Switch Ch2
        .CNC_A.LC_Ch1   // CNC3 Light Screen Ch1
        .CNC_A.DoorSW_Ch1   // CNC3 Door Switch Ch1
        .CNC_B.LC_Ch2   // CNC4 Light Screen Ch2
        .CNC_B.DoorSW_Ch2   // CNC4 Door Switch Ch2
        .CNC_B.LC_Ch1   // CNC4 Light Screen Ch1
        .CNC_B.DoorSW_Ch1   // CNC4 Door Switch Ch1
        .Perim.GateSW_Ch1   // Cell 2 Gate Switch Ch1
        .Perim.GateSW_Ch2   // Cell 2 Gate Switch Ch2
        .Perim.Ent_LC_Ch1   // Cell 2 Entry Light Screen Ch1
        .Perim.Ent_LC_Ch2   // Cell 2 Entry Light Screen Ch2
        .Perim.Exit_LC_Ch1   // Cell 2 Exit Light Screen Ch1
        .Perim.Exit_LC_Ch2   // Cell 2 Exit Light Screen Ch2
        .Perim.Ent_Mute1   // Entry Mute 1 (Mute Signals Inverted)
        .Perim.Ent_Mute2   // Entry Mute 2 (Mute Signals Inverted)
        .Perim.Exit_Mute1   // Exit Mute 1 (Mute Signals Inverted)
        .Perim.Exit_Mute2   // Exit Mute 2 (Mute Signals Inverted)
   C31DiverterHoldBack : PalletStop := (Ext := 1);
   C31PartInTransit : TIMER := (PRE := 11000);
   C3_Robot_ES_OK : BOOL := 1; {access None}
   C3_Robot_Gates_OK : BOOL := 1; {access None}
   C3EASRelay_Monitor : BOOL;   // Robot External Safety Gate Relay Monitor
   C3EESRelay_Monitor : BOOL;   // Robot External EStop Relay Monitor
   C3RobotStop : PalletStop := (Ret := 1);
   C3S : ABB_Cell_Safe := (Perim.GateSW_Ch1 := 1, Perim.GateSW_Ch2 := 1, Perim.Ent_LC_Ch1 := 1, Perim.Ent_LC_Ch2 := 1, Perim.Exit_LC_Ch1 := 1, Perim.Exit_LC_Ch2 := 1, Perim.Ent_Mute1 := 1, Perim.Ent_Mute2 := 1, Perim.Exit_Mute1 := 1, Perim.Exit_Mute2 := 1, Perim.EntMuteStatOK := 1, Perim.ExitMuteStatOK := 1, Perim.OK := 1, Perim.Ent_LC_Not_Blocked := 1, Perim.Exit_LC_Not_Blocked := 1);
        .Perim.Ent_Mute1   // Entry Mute 1 (Mute Signals Inverted)
        .Perim.Ent_Mute2   // Entry Mute 2 (Mute Signals Inverted)
        .Perim.Exit_Mute1   // Exit Mute 1 (Mute Signals Inverted)
        .Perim.Exit_Mute2   // Exit Mute 2 (Mute Signals Inverted)
   Camera1_Geometry2 : BOOL;
   Camera1_Geometry2_Dim : REAL := 12.513942;
   Camera1_Part_1_Distance : REAL := nan;
   Camera1_Part_1_Length : REAL := nan;
   Camera1_Part_1_Length_2 : REAL := nan;
   Camera1_Part_1_Width : REAL := nan;
   Camera1_Part_1_Width_2 : REAL := nan;
   Camera1_ZZ : TIMER := (PRE := 5000);
   Camera_RFID_Data_Test : SINT[4];
   Camera_RFID_Read_Test : SINT;
   Cell1_BadParts : COUNTER;
   Cell1_GoodParts : COUNTER;
   Cell1EntryLC : LIGHT_CURTAIN := (LCB := 1);   // Cell 1 Conveyor Entry Light Screen
   Cell1EntryLCMute : MUTING_TWO_SENSOR_SYM := (RestartType := 1, EnableMute := 1, InputStatus := 1, MutingLampStatus := 1, S1S2DiscrepancyTime := 1000, S1S2LCMinimumTime := 10, S1S2LCMaximumTime := 10000, MaximumMuteTime := 10, MaximumOverrideTime := 30, CA := 1, FP := 1, FaultCode := 36864);   // Celll 1 Entry LC Muting
   Cell1ExitLC : LIGHT_CURTAIN := (ChannelA := 1, ChannelB := 1, O1 := 1);   // Cell 1 Conveyor Exit Light Screen
   Cell1ExitLCMute : MUTING_TWO_SENSOR_SYM := (RestartType := 1, LightCurtain := 1, Sensor1 := 1, Sensor2 := 1, EnableMute := 1, InputStatus := 1, MutingLampStatus := 1, S1S2DiscrepancyTime := 1000, S1S2LCMinimumTime := 10, S1S2LCMaximumTime := 10000, MaximumMuteTime := 10, MaximumOverrideTime := 30, FP := 1, FaultCode := 39426);   // Celll 1 Exit LC Muting
   Cell1GateSW : REDUNDANT_INPUT := (ChannelA := 1, ChannelB := 1, O1 := 1);   // Cell 1 Entry Gate Switch
   Cell1PalletAtStop : BOOL;   // Part at Cell 1 Pallet Stop
   Cell2_BadParts : COUNTER;
   Cell2_GoodParts : COUNTER;
   Cell2EntryLC : LIGHT_CURTAIN := (ChannelA := 1, ChannelB := 1, MuteLightCurtain := 1, O1 := 1, LCM := 1);   // Cell 2 Conveyor Entry Light Screen
   Cell2EntryLCMute : MUTING_TWO_SENSOR_SYM := (RestartType := 1, LightCurtain := 1, Sensor1 := 1, Sensor2 := 1, EnableMute := 1, InputStatus := 1, MutingLampStatus := 1, S1S2DiscrepancyTime := 1000, S1S2LCMinimumTime := 10, S1S2LCMaximumTime := 10000, MaximumMuteTime := 10, MaximumOverrideTime := 30, O1 := 1);   // Celll 2 Entry LC Muting
   Cell2ExitLC : LIGHT_CURTAIN := (ChannelA := 1, ChannelB := 1, MuteLightCurtain := 1, O1 := 1, LCM := 1);   // Cell 2 Conveyor Exit Light Screen
   Cell2ExitLCMute : MUTING_TWO_SENSOR_SYM := (RestartType := 1, LightCurtain := 1, Sensor1 := 1, Sensor2 := 1, EnableMute := 1, InputStatus := 1, MutingLampStatus := 1, S1S2DiscrepancyTime := 1000, S1S2LCMinimumTime := 10, S1S2LCMaximumTime := 10000, MaximumMuteTime := 10, MaximumOverrideTime := 30, O1 := 1);   // Celll 2 Exit LC Muting
   Cell2GateSW : REDUNDANT_INPUT := (ChannelA := 1, ChannelB := 1, O1 := 1);   // Cell 2 Entry Gate Switch
   Cell3_BadParts : COUNTER;
   Cell3_GoodParts : COUNTER;
   Cell3EntryLC : LIGHT_CURTAIN := (ChannelA := 1, ChannelB := 1, O1 := 1);   // Cell 3 Conveyor Entry Light Screen
   Cell3EntryLCMute : MUTING_TWO_SENSOR_SYM := (RestartType := 1, LightCurtain := 1, Sensor1 := 1, Sensor2 := 1, EnableMute := 1, MutingLampStatus := 1, S1S2DiscrepancyTime := 500, S1S2LCMinimumTime := 10, S1S2LCMaximumTime := 1000, MaximumMuteTime := 3, MaximumOverrideTime := 15, DiagnosticCode := 32);   // Celll 3 Entry LC Muting
   Cell3ExitLC : LIGHT_CURTAIN := (ChannelA := 1, ChannelB := 1, O1 := 1);   // Cell 3 Conveyor Exit Light Screen
   Cell3ExitLCMute : MUTING_TWO_SENSOR_SYM := (RestartType := 1, LightCurtain := 1, Sensor1 := 1, Sensor2 := 1, EnableMute := 1, MutingLampStatus := 1, S1S2DiscrepancyTime := 500, S1S2LCMinimumTime := 10, S1S2LCMaximumTime := 1000, MaximumMuteTime := 3, MaximumOverrideTime := 15, DiagnosticCode := 32);   // Celll 3 Exit LC Muting
   Cell3GateSW : REDUNDANT_INPUT := (ChannelA := 1, ChannelB := 1, O1 := 1);   // Cell 3 Entry Gate Switch
   Cell_1 : Fanuc_Cell := (GoodParts.PRE := 32767, GoodParts.ACC := 475, RejectedParts.PRE := 32767, RejectedParts.ACC := 927);
   Cell_1_PartEntering : BOOL;   // Part in transit from hold back to robot stop
   Cell_2 : Fanuc_Cell := (GoodParts.PRE := 32767, GoodParts.ACC := 682, GoodParts.CU := 1, RejectedParts.PRE := 32767, RejectedParts.ACC := 591, RejectedParts.CU := 1);
   CellExitLCMute : MUTING_TWO_SENSOR_SYM;   // Celll 2 Exit LC Muting
   CircuitReset : BOOL;
   CircuitResetSafe : BOOL;   // Signal to Reset Circuits
   Clamp_To_Line : BOOL;
   Close_Clamp : BOOL;
   Cloud_R1Z_TagPresent : BOOL;
   Cloud_R1Z_Timer : TIMER := (PRE := 1000);
   Cloud_R2Z_TagPresent : BOOL;
   Cloud_R2Z_Timer : TIMER := (PRE := 1000);
   Cloud_R3Z_TagPresent : BOOL;
   Cloud_R3Z_Timer : TIMER := (PRE := 1000);
   Cloud_R4Z_TagPresent : BOOL;
   Cloud_R4Z_Timer : TIMER := (PRE := 1000);
   Cloud_R5Z_TagPresent : BOOL;
   Cloud_R5Z_Timer : TIMER := (PRE := 1000);
   Cloud_R6Z_TagPresent : BOOL;
   Cloud_R6Z_Timer : TIMER := (PRE := 1000);
   CNC1_Door : REDUNDANT_INPUT;   // CNC1 Door Switch
   CNC1_EStop : EMERGENCY_STOP := (ChannelA := 1, ChannelB := 1, O1 := 1);
   CNC1_LC : LIGHT_CURTAIN := (ChannelA := 1, ChannelB := 1, O1 := 1);   // CNC1 to Cell 1 Light Screen
   CNC1_ProcessTimer : TIMER := (PRE := 999999999, ACC := 1044269);
   CNC1_Switch_On : ALIAS FOR C2_N021:7:O.1;
   CNC1Bools : DINT;
   CNC1timer : SINT[4] := ([1] := -34, [2] := 15);
   CNC2_Door : REDUNDANT_INPUT := (ChannelA := 1, ChannelB := 1, O1 := 1);   // CNC2 Door Switch
   CNC2_EStop : EMERGENCY_STOP := (ChannelA := 1, ChannelB := 1, O1 := 1);
   CNC2_LC : LIGHT_CURTAIN := (ChannelA := 1, ChannelB := 1, MuteLightCurtain := 1, O1 := 1, LCM := 1);   // CNC2 to Cell 1 Light Screen
   CNC2_ProcessTimer : TIMER := (PRE := 999999999, ACC := 423637);
   CNC2Bools : DINT;
   CNC2timer : SINT[4] := ([0] := -43, [1] := 118, [2] := 6);   // Dint to Sint array
   CNC3_Door : REDUNDANT_INPUT;   // CNC3 Door Switch
   CNC3_EStop : EMERGENCY_STOP;
   CNC3_LC : LIGHT_CURTAIN := (ChannelA := 1, ChannelB := 1, O1 := 1);   // CNC3 to Cell 2 Light Screen
   CNC3_ProcessTimer : TIMER := (PRE := 999999999, ACC := 1044269);
   CNC3_Switch_On : BOOL;
   CNC3Bools : DINT;
   CNC3timer : SINT[4] := ([0] := 45, [1] := -17, [2] := 15);
   CNC4_Door : REDUNDANT_INPUT;   // CNC4 Door Switch
   CNC4_EStop : EMERGENCY_STOP := (ChannelA := 1, ChannelB := 1, O1 := 1);
   CNC4_LC : LIGHT_CURTAIN := (ChannelA := 1, ChannelB := 1, O1 := 1);   // CNC4 to Cell 2 Light Screen
   CNC4_ProcessTimer : TIMER := (PRE := 999999999, ACC := 423637);
   CNC4Bools : DINT;
   CNC4Simulator : TIMER := (PRE := 45000);
   CNC4timer : SINT[4] := ([0] := 122, [1] := 69, [2] := 6);
   CNC_1_Done : BOOL;   // CNC 1 has completed cutting the part
   CNC_1_idle : BOOL;
   CNC_1_ProgToRun : DINT := 4;
   CNC_1_Running : BOOL;
   CNC_2_Done : BOOL;   // CNC 2 has completed cutting the part
   CNC_2_idle : BOOL;
   CNC_2_ProgToRun : DINT := 2;   // G-Code Program Number for CNC to run TO CNC
   CNC_2_Running : BOOL;
   CNC_3_Done : BOOL;   // CNC 3 has completed cutting the part
   CNC_3_idle : BOOL := 1;
   CNC_3_ProgToRun : DINT := 4;   // G-code program number to be paassed to CNC to run
   CNC_3_Running : BOOL;
   CNC_4_Done : BOOL;   // CNC 4 has completed cutting the part
   CNC_4_idle : BOOL := 1;
   CNC_4_ProgToRun : DINT := 5;
   CNC_4_Running : BOOL;
   CNC_4_Timer : TIMER := (PRE := 500);
   CNC_4_ZZ : BOOL;
   CNC_idle : BOOL;
   CNC_On : BOOL := 1;
   Comm_Fault_Sts_Timer : TIMER;
   Comm_Fault_Sts_Timer1 : TIMER := (EN := 1, DN := 1);
   Comm_Fault_Sts_Timer2 : TIMER;
   Comm_Status : DINT;
   Comm_Status1 : DINT := 16384;
   Comm_Status2 : DINT := 16384;
   ContinuousRunCase : BOOL := 1;
   CountEmptyC2 : COUNTER := (DN := 1);
   Counter_Drop_CNC1 : COUNTER := (PRE := 1);   // Countes when the robot has droped a part at CNC1
   Counter_Pick_Conv : COUNTER := (PRE := 1, ACC := 5, DN := 1);   // Counts when the robot has picked a part from conveyor
   DatacollectTry : INT;
   DataTryRF : SINT;
   DeBounce1 : TIMER := (PRE := 250);
   DeBounce2 : TIMER := (PRE := 250);
   DeBounce3 : TIMER := (PRE := 250);
   DeBounce4 : TIMER := (PRE := 250);
   DeBounce5 : TIMER := (PRE := 1000);
   DeBounce6 : TIMER := (PRE := 2000);
   DeBounce7 : TIMER := (PRE := 2000);
   DeBounce8 : TIMER := (PRE := 2000);
   DeBounceC23DivHoldBack : TIMER := (PRE := 1000);
   dest01 : SINT[10] := ([0] := -35, [1] := -52, [2] := -69, [3] := -86);
   detect_4 : BOOL;
   Drop_CNC1 : BOOL;   // Send signal to drop part at CNC1
   Drop_CNC2 : BOOL;   // Send signal to drop part at CNC2
   Drop_Conv : BOOL;   // Send signal to drop part at conveyor
   Dry_Cycle : BOOL;
   Dry_Cycle_Safe : BOOL;
   DryCycleDelay2 : TIMER := (PRE := 5000);
   DryCycleDelay4 : TIMER := (PRE := 5000);
   Empty_pallet : BOOL;
   EmptyStart : TIMER := (PRE := 500);
   Enable_Cell_3 : BOOL;   // Turn bit on to enable logic for Cell 3
   Enable_CNC1 : BOOL := 1;
   Enable_CNC2 : BOOL := 1;
   Enable_CNC3 : BOOL := 1;
   Enable_CNC4 : BOOL := 1;
   Enable_Process_Update : BOOL;
   EnableBits : DINT := 63;
   Extend_Stop : BOOL;
   Fanuc_Loop_Conv_ES_Ch1 : BOOL := 1;   // Cell 1/2 Conveyor Pull Cord / E-Stop Ch1
   Fanuc_Loop_Conv_ES_Ch2 : BOOL := 1;   // Cell 1/2 Conveyor Pull Cord / E-Stop Ch2
   Fanuc_Loop_Conv_Safety_OK : BOOL := 1;
   Fanuc_Loop_Speed : DINT;
   FanucLoopPullCordES : EMERGENCY_STOP := (ChannelA := 1, ChannelB := 1, O1 := 1);   // EStop / Cable On Fanuc Loop
   FanucLoopPullCordESCH1 : BOOL;   // Cell 1/2 pull Cord CH1
   FanucLoopPullCordESCH2 : BOOL;   // Cell 1/2 pull Cord CH2
   FanucLoopSTO_O1 : BOOL := 1;
   FanucLoopSTO_O2 : BOOL := 1;
   FanucLoopVFD : PF525_Faceplate_AOI := (Inp_NumRowsVis := 9, Sts_ProgramModeEnabled := 1, Sts_DriveStatus_Faulted := 1, Sts_DriveStatus_ActualDir := 1, Sts_DeviceState := 2, Set_Value1Max := 60, Set_Value2Max := 1, Set_Value3Max := 1, Val_TrendMax := 60, Val_Fault1Code := 52073, Cmd_OperToProgPermissive := 1, Cmd_ProgToOperPermissive := 1, Set_SpeedOper := 30, Set_CommFaultTimerPresetProg := 10000, Set_SpeedProg := 30, Set_DecelOper := 1.5, Set_AccelOper := 1.5, Comm_Status := 16384, Inst_Error := 1, LastFaultCode := 73, SpdRef_Units := 30, SpdScaler60Hz := 1.0, GearRatio := 1.0, Out_SpdRef_Units := 30, Sts_PowerflexAlarmTrigger := 52073);
   fault_code : DINT;
   Fault_Code1 : DINT := 73;
   Fault_Code2 : DINT := 105;
   Fault_Msg : MESSAGE;
        MessageParameters(ServiceCode := 16#000e, DestinationTag := fault_code, ...)
   FaultReset : BOOL;
   FaultResetSafe : BOOL;
   Fest03 : DINT;
   Festo_Air_On : BOOL := 1;
   FestoAI0 : DINT := 2;
   FestoAI1 : DINT;
   FestoAI2 : DINT;
   FestoAI3 : DINT;
   FestoAIP0 : DINT := 140;
   FestoAIP1 : DINT := 140;
   FestoAIP2 : DINT := 100;
   FestoAIP3 : DINT := 160;
   Fetching_matl : BOOL;
   FltMsg1 : MESSAGE;
        MessageParameters(ServiceCode := 16#000e, DestinationTag := Fault_Code1, ...)
   FltMsg2 : MESSAGE;
        MessageParameters(ServiceCode := 16#000e, DestinationTag := Fault_Code2, ...)
   FromCNC1 : CNC_Datablock := (Bools := 32);   // Data From CNC1
        .Bools.0   // CNC signal to Cell that it is at the Pick / Drop location
        .Bools.1   // CNC is ready to receive part from robot
        .Bools.2   // Handshake to complete part drop off
        .Bools.3   // CNC has a part that is ready to be picked up by the robot
        .Bools.4   // Handshake to complete part Pick-up
   FromCNC2 : CNC_Datablock := (Bools := 32);   // Data From CNC2
        .Bools.0   // CNC signal to Cell that it is at the Pick / Drop location
        .Bools.1   // CNC is ready to receive part from robot
        .Bools.2   // Handshake to complete part drop off
        .Bools.3   // CNC has a part that is ready to be picked up by the robot
        .Bools.4   // Handshake to complete part Pick-up
   FromCNC3 : CNC_Datablock := (Bools := 32);   // Data From CNC3
        .Bools.0   // CNC signal to Cell that it is at the Pick / Drop location
        .Bools.1   // CNC is ready to receive part from robot
        .Bools.2   // Handshake to complete part drop off
        .Bools.3   // CNC has a part that is ready to be picked up by the robot
        .Bools.4   // Handshake to complete part Pick-up
        .Bools.5   // Bit is ON when CNC is NOT in cycle.
   FromCNC4 : CNC_Datablock := (Bools := 32);   // Data From CNC4
        .Bools.0   // CNC signal to Cell that it is at the Pick / Drop location
        .Bools.1   // CNC is ready to receive part from robot (M72)
        .Bools.2   // Handshake to complete part drop off
        .Bools.3   // CNC has a part that is ready to be picked up by the robot (M73)
        .Bools.4   // Handshake to complete part Pick-up
        .Bools.5   // Bit is ON when CNC is NOT in cycle.
   Gantry_busy : BOOL;
   Gantry_prep : BOOL;
   Gantry_reload : BOOL := 1;
   Gantry_start : BOOL;
   gjf : BOOL;
   Go_Home : BOOL;   // Send signal to go to pounce
   HMI_Disp_No : DINT := 600;
   HMI_Mode : DINT;
   HMI_Stop_Fan_Loop_VFD : BOOL;
   HMI_Strt_Fan_Loop_VFD : BOOL;
   Holding_matl : BOOL;
   Horoz_Adv : BOOL;
   ImageFail : BOOL;
   ImagePass : BOOL;
   InstaceTEST : DINT;
   Jumper : BOOL := 1;
   JumperS : BOOL := 1;
   Lower_Slide : BOOL;
   MainPnlES : EMERGENCY_STOP := (ChannelA := 1, ChannelB := 1, O1 := 1);   // EStop on Main Panel
   MainPnlESCH1 : BOOL := 1;   // Main Panel E-Stop Button CH1
   MainPnlESCH2 : BOOL := 1;   // Main Panel E-Stop Button CH2
   Man_Valves : DINT[8] := ([0] := 1, [1] := 1, [2] := 1, [3] := 1, [4] := 1, [6] := 1, [7] := 1);
   Man_Valves01 : SINT := -86;
   Man_Valves02 : SINT := -90;
   Man_Valves_Safe01 : SINT := -103;
   Man_Valves_Safe02 : SINT := 85;
   Matl_delivered : BOOL := 1;
   Mode_Auto : BOOL;
   Mode_Auto_Safe : BOOL;
   Mode_Manual : BOOL;
   Mode_Manual_Safe : BOOL;
   Mode_None : BOOL := 1;
   Mode_None_Safe : BOOL := 1;
   Mode_Semi : BOOL;
   Mode_Start : BOOL;
   Move_Conv_RawMat : BOOL := 1;
   Move_Cov_RawMat : BOOL;
   NI_1752_Camera : MESSAGE;
   ONS : DINT := 2228504;
   Open_Clamp : BOOL := 1;
   PaletClearPreset : DINT[8] := ([0] := 700, [1] := 600, [2] := 700, [3] := 600, [4] := 450, [5] := 1000, [6] := 1000, [7] := 1000);
   PalletAtC2C3HoldBack : BOOL;   // Pallet at Cell 2 to Cell 3 Diverter Hold Back Stop
   Part1_Distance : STRING := 'nan';
   Part1_Length1 : STRING := 'nan';
   Part1_Length2 : STRING := 'nan';
   Part1_Width1 : STRING := 'nan';
   Part1_Width2 : STRING := 'nan';
   Part_A : BOOL;
   Part_A_input : COUNTER := (ACC := 7, DN := 1);
   Part_A_output : COUNTER := (DN := 1);
   Part_B : BOOL;
   Part_B_input : COUNTER := (ACC := 4, DN := 1);
   Part_B_output : COUNTER := (DN := 1);
   Part_dropped : BOOL := 1;
   Part_from_conv_holding : BOOL;
   Part_ready_for_Gantry : BOOL;
   PF525 : PF525_Faceplate_AOI := (Inp_NumRowsVis := 9, Set_Value1Max := 60, Set_Value2Max := 1, Set_Value3Max := 1, Cmd_OperToProgPermissive := 1, Cmd_ProgToOperPermissive := 1, Set_CommFaultTimerPresetProg := 10000);
   PF525_AlarmName : STRING;
   PF525_AlarmName1 : STRING;
   PF525_AlarmName2 : STRING;
   PF525_FaultCodeList : P_DescList[61] := ([0].Desc := 'Check drive manual for this fault code', [1].Code := 2, [1].Desc := 'Auxiliary Input', [2].Code := 3, [2].Desc := 'Power Loss', [3].Code := 4, [3].Desc := 'Under Voltage', [4].Code := 5, [4].Desc := 'Over Voltage', [5].Code := 6, [5].Desc := 'Motor Stalled', [6].Code := 7, [6].Desc := 'Motor Overload', [7].Code := 8, [7].Desc := 'Heatsink Overtemp', [8].Code := 9, [8].Desc := 'CC OverTemp', [9].Code := 12, [9].Desc := 'Hardware Overcurrent', [10].Code := 13, [10].Desc := 'Ground Fault', [11].Code := 15, [11].Desc := 'Load Loss', [12].Code := 21, [12].Desc := 'Output Phase Loss', [13].Code := 29, [13].Desc := 'Analog Input Loss', [14].Code := 33, [14].Desc := 'Auto Restart Tries', [15].Code := 38, [15].Desc := 'Phase U to Ground', [16].Code := 39, [16].Desc := 'Phase V to Ground', [17].Code := 40, [17].Desc := 'Phase W to Ground', [18].Code := 41, [18].Desc := 'Phase U-V Short', [19].Code := 42, [19].Desc := 'Phase U-W Short', [20].Code := 43, [20].Desc := 'Phase V-W Short', [21].Code := 48, [21].Desc := 'Parameters Defaulted', [22].Code := 59, [22].Desc := 'Safety Open', [23].Code := 63, [23].Desc := 'SW Over Current', [24].Code := 64, [24].Desc := 'Drive Overload', [25].Code := 70, [25].Desc := 'Power Unit', [26].Code := 71, [26].Desc := 'DSI Net Loss', [27].Code := 72, [27].Desc := 'Opt Net Loss', [28].Code := 73, [28].Desc := 'Ethernet Net Loss', [29].Code := 80, [29].Desc := 'AutoTune Failure', [30].Code := 81,
        [30].Desc := 'DSI Comm Loss', [31].Code := 82, [31].Desc := 'Opt Comm Loss', [32].Code := 83, [32].Desc := 'Ethernet Comm Loss', [33].Code := 91, [33].Desc := 'Encoder Loss', [34].Code := 94, [34].Desc := 'Function Loss', [35].Code := 100, [35].Desc := 'Parameter Checksum', [36].Code := 101, [36].Desc := 'External Storage', [37].Code := 105, [37].Desc := 'C Connect Error', [38].Code := 106, [38].Desc := 'Incompat. C-P', [39].Code := 107, [39].Desc := 'Replaced C-P', [40].Code := 109, [40].Desc := 'Mismatch C-P', [41].Code := 110, [41].Desc := 'Keypad Membrane', [42].Code := 111, [42].Desc := 'Safety Hardware', [43].Code := 114, [43].Desc := 'uC Failure', [44].Code := 122, [44].Desc := 'I/O Baord Fail', [45].Code := 125, [45].Desc := 'Flash Update Reqd', [46].Code := 126, [46].Desc := 'Unrecoverable Error', [47].Code := 127, [47].Desc := 'DSI Flash Update Reqd');   // PowerFlex 525 VFD Fault Codes and Descriptions
   PF_525I : AB:PowerFlex525V_E_8A02D441:I:0;
   PF_525O : AB:PowerFlex525V_E_5483BAFD:O:0;
   Pick_CNC1 : BOOL;   // Send signal to pick part from CNC1
   Pick_CNC2 : BOOL;   // Send signal to pick part from CNC2
   Pick_Conv : BOOL;   // Send signal to pick part from conveyor
   Picking_up_part : BOOL;
   PLC_Day : DINT := 8;
   PLC_Hour : DINT := 2;
   PLC_Microsecond : DINT := 772208;
   PLC_Minute : DINT := 48;
   PLC_Month : DINT := 10;
   PLC_Second : DINT := 1;
   PLC_Time : DINT[7] := ([0] := 1998, [1] := 10, [2] := 8, [3] := 2, [4] := 48, [5] := 2, [6] := 372207);
   PLC_Year : DINT := 1998;
   PowerFlexAlarmName : STRING;
   PowerFlexAlarmName1 : STRING;
   PowerFlexAlarmName2 : STRING;
   PowerFlexAlarmTrigger : DINT;
   PowerFlexAlarmTrigger1 : DINT;
   PowerFlexAlarmTrigger2 : DINT;
   PPX1 : ALIAS FOR C1_N011:6:I.7;   // Sensor Palet Stop RFID1 (Cell 1 Fanuc Robot Stop)
   PPX2 : ALIAS FOR Conv_N053:3:I.0;   // Sensor Pallet Stop RFID2 (Cell 2 Hold Back Stop)
   PPX3 : ALIAS FOR Conv_N053:3:I.1;   // Sensor Pallet Stop RFID3 (Cell 2 Fanuc Robot Stop)
   PPX4 : ALIAS FOR Conv_N053:3:I.2;   // Sensor Pallet Stop RFID4 (Loop 1 Diverter Hold Back Stop)
   PPX5 : ALIAS FOR Main_N043:3:I.0;   // Sensor Pallet Stop (Cell 1 Hold Back)
   PPX6 : ALIAS FOR C3_N031:5:I.1;   // Sensor Pallet Stop RFID6 (Loop 2 Diverter Hold Back Stop)
   PPX7 : ALIAS FOR C3_N031:5:I.0;   // Sensor Pallet Stop RFID7 (Cell 3 ABB Robot Stop)
   R1J_Assign : BOOL;
   R1J_Check_Process_NO : DINT := 1;
   R1J_Current_Part_NO : SINT := 2;
   R1J_Current_Process_NO : SINT := 3;
   R1J_Process : BOOL := 1;
   R1J_Read : BOOL;
   R1J_Read_Check_Fail : BOOL;
   R1J_Read_Check_InProgress : BOOL;
   R1J_Read_Check_Results : BOOL;
   R1J_Read_Check_Start : BOOL;
   R1J_Read_Finished : BOOL;
   R1J_Read_InProgress : BOOL;
   R1J_Read_Results : BOOL;
   R1J_Read_Start : BOOL;
   R1J_Write : BOOL;
   R1J_Write_Finished_Check : BOOL;
   R1J_Write_Inprogress : BOOL;
   R1J_Write_Pass : BOOL;
   R1Z_Pass : BOOL;
   R2Z_Current_Part_NO : DINT := 2;
   R2Z_Current_Process_NO : DINT := 3;
   R2Z_Read : BOOL;
   R2Z_Read_Finished : BOOL;
   R2Z_Read_InProgress : BOOL;
   R2Z_Read_Results : BOOL;
   R2Z_Read_Start : BOOL;
   R3J_Assign : BOOL;
   R3J_Check_Process_NO : DINT := 2;
   R3J_Current_Part_NO : SINT := 2;
   R3J_Current_Process_NO : SINT := 3;
   R3J_Process : BOOL;
   R3J_Read : BOOL;
   R3J_Read_Check_Fail : BOOL;
   R3J_Read_Check_InProgress : BOOL;
   R3J_Read_Check_Results : BOOL;
   R3J_Read_Check_Start : BOOL;
   R3J_Read_Finished : BOOL;
   R3J_Read_InProgress : BOOL;
   R3J_Read_Results : BOOL;
   R3J_Read_Start : BOOL;
   R3J_Write : BOOL;
   R3J_Write_Finished_Check : BOOL;
   R3J_Write_Inprogress : BOOL;
   R3J_Write_Pass : BOOL;
   R5Z_Current_Part_NO : DINT := 2;
   R5Z_Current_Process_NO : DINT := 3;
   R5Z_Read : BOOL;
   R5Z_Read_Finished : BOOL;
   R5Z_Read_InProgress : BOOL;
   R5Z_Read_Results : BOOL;
   R5Z_Read_Start : BOOL;
   R6S_Check_Current_Part_NO : DINT := 2;
   R6S_Check_Current_Process_NO : DINT;
   R6S_User_Input_Part_NO : DINT := 2;
   R6S_User_Input_Process_NO : DINT;
   R6Z_Check_Read_PB : BOOL;
   R6Z_Check_Write : BOOL;
   R6Z_Clear_All_PB : BOOL;
   R6Z_Clear_Mode : BOOL;
   R6Z_Clear_Mode_PB : BOOL;
   R6Z_Write_Check : BOOL;
   R6Z_Write_Check_1 : BOOL;
   R6Z_Write_Inprogress_Check : BOOL;
   R6Z_Write_Inprogress_Check_1 : BOOL;
   R6Z_Write_Test : BOOL;
   R6Z_Write_Test_1 : BOOL;
   R6Z_Write_Test_PB : BOOL;
   Raise_Slide : BOOL := 1;
   REAL_test : REAL;
   RelC1HoldBack : TIMER := (PRE := 700);
   RelC1RobotStop : TIMER := (PRE := 600);
   RelC2HoldBack : TIMER := (PRE := 700);
   RelC2RobotStop : TIMER := (PRE := 600);
   resetC2RobTimer : TIMER := (PRE := 1000);
   Return_Slide : BOOL;
   RFID1timer : SINT[4];
   RFID2timer : SINT[4];   // DINT to SINT
        [0]   // DINT to SINT
   RFID4timer : SINT[4];
   RFID5timer : SINT[4];
   RFID6timer : SINT[4];
   RFID_ReadData1 : SINT;
   RFID_ReadData1p : SINT;
   RFID_ReadData1p1 : SINT;
   RFID_ReadData1process : DINT;
   RFID_ReadData1processtime : DINT;
   RFID_ReadData1timer : SINT[4];
   RFID_ReadData2 : SINT;
   RFID_ReadData2p : SINT;
   RFID_ReadData2process : DINT;
   RFID_ReadData2processtime : DINT;
   RFID_ReadData2timer : SINT[4];
   RFID_ReadData3 : SINT := 1;
   RFID_ReadData3p : DINT;
   RFID_ReadData3process : DINT := 1;
   RFID_ReadData3processtime : DINT;
   RFID_ReadData3timer : SINT[4] := ([0] := -43, [1] := 118, [2] := 6);
   RFID_ReadData4 : SINT;
   RFID_ReadData4p : SINT;
   RFID_ReadData4process : DINT;
   RFID_ReadData4processtime : DINT;
   RFID_ReadData4timer : SINT[4];
   RFID_ReadData5 : SINT;
   RFID_ReadData5p : DINT;
   RFID_ReadData5process : DINT;
   RFID_ReadData5processtime : DINT;
   RFID_ReadData5timer : SINT[4];
   RFID_ReadData6 : SINT;
   RFID_ReadData6p : SINT;
   RFID_ReadData6process : SINT;
   RFID_ReadData6processtime : DINT;
   RFID_ReadData6timer : SINT[4];
   RFID_ReadData7 : SINT;
   RFID_ReadData_2 : SINT;   // Will store data read from the tag
   RFID_ReadData_4 : SINT;
   RFID_Write_1 : BOOL := 1;
   RFID_Write_2 : BOOL := 1;
   RFID_Write_3 : BOOL := 1;
   RFID_Write_4 : BOOL := 1;
   RFID_Write_5 : BOOL := 1;
   RFID_Write_6 : BOOL := 1;
   RFID_Write_Byte_Start_1 : BOOL;
   RFID_Write_Byte_Start_2 : BOOL := 1;
   RFID_Write_Byte_Start_3 : BOOL;
   RFID_Write_Byte_Start_4 : BOOL;
   RFID_Write_Byte_Start_5 : BOOL;
   RFID_Write_Byte_Start_6 : BOOL;
   RFID_Write_InProgress : BOOL;
   RFID_Write_inProgress4 : BOOL;
   RFID_WriteData1 : SINT := 1;
   RFID_WriteData1p : SINT := 96;
   RFID_WriteData2 : SINT := 4;
   RFID_WriteData3 : SINT := 3;
   RFID_WriteData3p : SINT := 97;
   RFID_WriteData4 : SINT := 4;
   RFID_WriteData5 : SINT := 5;
   RFID_WriteData6 : SINT := 6;
   RFID_WriteData7 : SINT;
   RFID_WriteData_2 : SINT := 7;   // Stores data to be written to object
   RFID_WriteData_3 : SINT := 2;
   RFID_WriteData_4 : SINT;
   RFID_WriteData_5 : SINT := 4;
   RFID_WritePartA : SINT := 96;
   RFID_WritePartB : SINT := 97;
   RFID_WritePartC : SINT := 98;
   RFID_WriteProcess0 : DINT;
   RFID_WriteProcess1 : DINT := 1;
   RFID_WriteProcess2 : DINT := 2;
   RFID_WriteProcess3 : DINT := 2;
   RFID_WriteProcess4 : DINT := 2;
   RFIDTP1 : ALIAS FOR RFID_N054:I.Channel[0].TagPresent;   // RFID Tag at Cell 1 Stop
   RFIDTP2 : ALIAS FOR RFID_N054:I.Channel[1].TagPresent;   // RFID Tag at Cell 2 Hold Back Stop
   RFIDTP3 : ALIAS FOR RFID_N055:I.Channel[0].TagPresent;   // RFID Tag at Cell 2 Stop
   RFIDTP4 : ALIAS FOR RFID_N055:I.Channel[1].TagPresent;   // RFID Tag at Cell C23 Hold Back Stop
   RFIDTP5 : ALIAS FOR RFID_N056:I.Channel[0].TagPresent;   // RFID Tag at Cell 3 Stop
   RFIDTP6 : ALIAS FOR RFID_N056:I.Channel[1].TagPresent;
   Robot1_Busy_ZZ : BOOL;
   Robot1_CarryingPart : BOOL;
   Robot1_DroppedP1 : BOOL;
   Robot1_DroppedP2 : BOOL;
   Robot1_Flipped : BOOL;
   Robot1DroppedPart : BOOL;
   Robot2_Busy_ZZ : BOOL;
   Robot2_CarryingPart : BOOL;
   Robot2_Dropped3 : BOOL;
   Robot2_DroppedP3 : BOOL;
   Robot2_DroppedP4 : BOOL;
   Robot2_Idle_ZZ : BOOL;
   Robot2DroppedPart : BOOL;
   Robot_DroppedP1 : BOOL;
   Run_gantry_logic : BOOL := 1;
   RunABBLoopatSpeed : BOOL;
   RunASynchCase : BOOL;
   RunCont : BOOL;
   RungCommentS : BOOL := 1;
   Running : BOOL := 1;
   RunPartOnCNC1 : BOOL;
   RunPartOnCNC2 : BOOL;
   RunpartOnCNC3 : BOOL;
   RunPartOnCNC4 : BOOL;
   RunSynch : BOOL;
   RunSynchCase : BOOL := 1;
   SC105 : P_PF52x := (Inp_FwdPermOK := 1, Inp_FwdNBPermOK := 1, Inp_RevPermOK := 1, Inp_RevNBPermOK := 1, Inp_IntlkOK := 1, Inp_NBIntlkOK := 1, Cfg_SetTrack := 1, Cfg_PCmdClear := 1, Cfg_ShedOnFailToStart := 1, Cfg_ShedOnIOFault := 1, Cfg_FailToStartAckReqd := 1, Cfg_FailToStopAckReqd := 1, Cfg_IntlkTripAckReqd := 1, Cfg_DriveFaultAckReqd := 1, Cfg_IOFaultAckReqd := 1, Cfg_FailToStartSeverity := 1000, Cfg_FailToStopSeverity := 1000, Cfg_IntlkTripSeverity := 500, Cfg_DriveFaultSeverity := 1000, Cfg_IOFaultSeverity := 1000, Cfg_MaxSpdRef := 60.0, Cfg_SpeedRefRawMax := 6000, Cfg_SpeedRefEUMax := 60.0, Cfg_SpeedFdbkRawMax := 6000, Cfg_SpeedFdbkEUMax := 60.0, Cfg_SimRampT := 10, Cfg_FailToStartT := 15, Cfg_FailToStopT := 15, Cfg_ResetPulseT := 2, Val_SpeedRefEUMax := 60.0, Val_SpeedFdbkEUMax := 60.0, Val_OutPower := 24.0, Val_Fault := 18, Val_Mode := 9, Sts_ActualDir := 1, Ack_FailToStart := 1, Ack_FailToStop := 1, Ack_IntlkTrip := 1, Ack_DriveFault := 1, Ack_IOFault := 1);   // Pump 105 Motor (PowerFlex 525 drive)
   SensosorPalletstopC23 : BOOL;
   SimulateCNC4 : BOOL;
   so_AcceptMSG00 : MESSAGE;
        MessageParameters(ServiceCode := 16#0050, LocalElement := so_OpenParams.Timeout, DestinationTag := so_AcceptResponse, ...)
   so_AcceptResponse : AcceptResponse := (Addr.Family := 2, Addr.Port := 11000);
   so_CreateInstance : DINT;
   so_CreateMSG00 : MESSAGE;
        MessageParameters(ServiceCode := 16#004b, LocalElement := so_CreateParams, DestinationTag := so_CreateInstance, ...)
   so_CreateParams : AcceptResponse := (Addr.Family := 2, Addr.Port := 11000);
   so_OpenMSG00 : MESSAGE;
        MessageParameters(ServiceCode := 16#004c, LocalElement := so_OpenParams, ...)
   so_OpenParams : OpenConnParams := (Timeout := 10000, DestAddr := '192.168.1.74?port=11000');
   Step_000 : SFC_STEP := (Status := 16#0020_0000, PauseTimer := 1);
   t1 : TIMER := (PRE := 5000);
   t11 : TIMER := (PRE := 5000);
   test01 : DINT := -1430532899;
   test02 : DINT := -1430532899;
   Test_String : STRING := '13.7122736';
   Test_String2 : STRING := '12.5139418';
   Test_ZZ : BOOL := 1;
   Test_ZZ_Good : BOOL;
   TestBedOptions : DINT;
   testrhu : DINT;
   Timer_RFID1 : TIMER := (PRE := 2000);
   Timer_RFID2 : TIMER;
   Timer_RFID21 : TIMER := (PRE := 2000);
   Timer_RFID3 : TIMER := (PRE := 2000);
   Timer_RFID4 : TIMER := (PRE := 2000);
   Timer_RFID4_W : TIMER := (PRE := 200);
   Timer_RFID5 : TIMER := (PRE := 2000);
   Timer_RFID6_Read : TIMER := (PRE := 3000);
   Timer_RFID7 : TIMER;
   Timer_RFIDt1 : TIMER := (PRE := 5000);
   Timer_RFIDt2 : TIMER := (PRE := 5000);
   TimerG1 : TIMER := (PRE := 2000);
   TimerG2 : TIMER := (PRE := 2000);
   TimerG3 : TIMER := (PRE := 2000);
   TimerG4 : TIMER := (PRE := 2000);
   TimerG5 : TIMER := (PRE := 2000);
   TimerG6 : TIMER := (PRE := 2000);
   TimerG7 : TIMER := (PRE := 2000);
   TimerG8 : TIMER := (PRE := 1000);
   TIMERON : TIMER := (PRE := 3000);
   TIMERON1 : TIMER := (PRE := 2000);
   TIMERON2 : TIMER := (PRE := 3000);
   TIMERON3 : TIMER := (PRE := 3000);
   TIMERON4 : TIMER := (PRE := 3000);
   TIMERON5 : TIMER := (PRE := 3000);
   TIMERON6 : TIMER := (PRE := 3000);
   ToCNC1 : CNC_Datablock := (UserDef01 := 4); {produced}   // Data To CNC1
        .UserDef01   // G-Code Program Number for CNC to run TO CNC
        .Bools.0   // Part Drop Request Cell (Robot) wants to load a part into the CNC
        .Bools.1   // Robot is clear of CNC - Drop or Pick is complete
        .Bools.31   // Set to 1 for Main Cell controller to pick program to run
   ToCNC2 : CNC_Datablock := (UserDef01 := 2); {produced}   // Data To CNC2
        .UserDef01   // G-Code Program Number for CNC to run TO CNC
        .Bools.0   // Part Drop Request Cell (Robot) wants to load a part into the CNC
        .Bools.1   // Robot is clear of CNC - Drop or Pick is complete
        .Bools.31   // Set to 1 for Main Cell controller to pick program to run
   ToCNC3 : CNC_Datablock := (UserDef01 := 4); {produced}   // Data To CNC3
        .UserDef01   // G-Code Program Number for CNC to run TO CNC
        .Bools.0   // Part Drop Request Cell (Robot) wants to load a part into the CNC
        .Bools.1   // Robot is clear of CNC - Drop or Pick is complete
        .Bools.31   // Set to 1 for Main Cell controller to pick program to run
   ToCNC4 : CNC_Datablock := (UserDef01 := 5); {produced}   // Data To CNC4
        .UserDef01   // G-Code Program Number for CNC to run TO CNC
        .Bools.0   // Part Drop Request Cell (Robot) wants to load a part into the CNC
        .Bools.1   // Robot is clear of CNC - Drop or Pick is complete
        .Bools.31   // Set to 1 for Main Cell controller to pick program to run
   Tran_000 : BOOL;
   Trigger_RFID_Read_2 : BOOL;
   Triggers : DINT;
   Unused_S_In : BOOL;   // Tag to indicate bit is unused in I/O mapping
   Unused_S_Out : BOOL;   // Unused Safety Output - Replace as needed
   Vac_On : BOOL;
   Vac_To_Line : BOOL := 1;
   ValvesOff : SINT;
   VFDFanucLoop_I : P_PF52x_Inp := (DriveStatus := 2#0000_0110_1000_1100, DriveStatus_CommandDir := 1, DriveStatus_ActualDir := 1, DriveStatus_Faulted := 1, DriveStatus_CommFreqCnt := 1, DriveStatus_CommLogicCnt := 1, OutputPower := 2400);
   VFDFanucLoop_O : P_PF52x_Out;
   ZZ_String : STRING;
   ZZ_String_2 : SINT;
   ZZ_Test : BOOL;
END_VAR

PROGRAM Data_Collection   (* main routine Main *)

ROUTINE Main   (* ladder *)
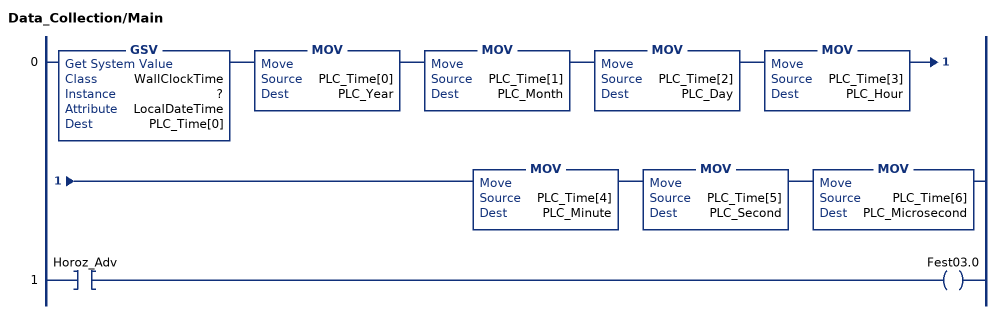
   0: GSV(WallClockTime,?,LocalDateTime,PLC_Time[0])MOV(PLC_Time[0],PLC_Year)MOV(PLC_Time[1],PLC_Month)MOV(PLC_Time[2],PLC_Day)MOV(PLC_Time[3],PLC_Hour)MOV(PLC_Time[4],PLC_Minute)MOV(PLC_Time[5],PLC_Second)MOV(PLC_Time[6],PLC_Microsecond);
   1: XIC(Horoz_Adv)OTE(Fest03.0);
END_ROUTINE
END_PROGRAM

PROGRAM MainProgram   (* main routine MainRoutine *)
VAR
   C23EmptyPalet : TIMER := (PRE := 1000);
   Camera1_Geometry1 : BOOL;
   Camera1_Geometry1_Dim : REAL := 13.712274;
   Camera1_Geometry1_Dim_Read : REAL;
   Camera1_Geometry1_Read : BOOL;
   Camera2_Geometry1 : BOOL;
   Camera2_Geometry1_Dim : REAL;
   Camera2_Geometry1_Dim_Read : REAL;
   Camera2_Geometry1_Read : BOOL;
   Camera_1_Trigger : BOOL;
   Camera_2_Trigger : BOOL;
   Clear_Multiple_Bytes : BOOL;
   Clear_Multiple_Bytes_InProgress : BOOL;
   Clear_Multiple_Bytes_Start : BOOL;
   Counter_1 : COUNTER := (ACC := 2549, DN := 1);
   Detect_2 : BOOL;
   DSFID_Value : DINT := 84;
   Enable_Clear_Multiple_Bytes : BOOL;
   HMI_Write_on : BOOL;
   HMI_WritePart : DINT := 96;
   L1 : BOOL;
   L2 : BOOL;
   L3 : BOOL;
   mtime : TIMER := (PRE := 1000);
   Part_Type_Counter : SINT := 2;
   Partintransittodiv : BOOL;
   Partintransittodiverter : TIMER := (PRE := 8000);
   PlaceKeeper : BOOL;
   R6Z_Assign : BOOL;
   R6Z_Check_Current : DINT := 3;
   R6Z_Check_Current1 : DINT;
   R6Z_Check_InProgress : BOOL;
   R6Z_Check_Part_NO : SINT := 3;
   R6Z_Check_Read : BOOL;
   R6Z_Check_Results : BOOL;
   R6Z_Check_Start : BOOL;
   R6Z_Clear_All : BOOL;
   R6Z_Clear_All_Inprogress : BOOL;
   R6Z_Clear_All_Start : BOOL;
   R6Z_Current_Part_NO : SINT := 3;
   R6Z_Current_Process_NO : SINT := 3;
   R6Z_Part_Type_Counter : SINT := 3;
   R6Z_Process : BOOL;
   R6Z_Read : BOOL;
   R6Z_Read_Check_Fail : BOOL;
   R6Z_Read_Check_InProgress : BOOL;
   R6Z_Read_Check_Results : BOOL;
   R6Z_Read_Check_Start : BOOL;
   R6Z_Read_Finished : BOOL;
   R6Z_Read_InProgress : BOOL;
   R6Z_Read_Results : BOOL;
   R6Z_Read_Start : BOOL;
   R6Z_Set_Part_Type : BOOL;
   R6Z_Write : BOOL;
   R6Z_Write_Finished_Check : BOOL;
   R6Z_Write_Inprogress : BOOL;
   R6Z_Write_Pass : BOOL;
   Read_InProgress : BOOL;
   RFID_Address : DINT;
   RFID_BlockSize : DINT;
   RFID_Length : DINT := 17;
   RFID_Read : BOOL;
   RFID_Read6_1_finished : BOOL;
   RFID_Read6_2_finished : BOOL;
   RFID_Read_1 : BOOL := 1;
   RFID_Read_2 : BOOL := 1;
   RFID_Read_3 : BOOL := 1;
   RFID_Read_4 : BOOL := 1;
   RFID_Read_5 : BOOL := 1;
   RFID_Read_6 : BOOL := 1;
   RFID_Read_Byte_Start_1 : BOOL := 1;
   RFID_Read_Byte_Start_2 : BOOL;
   RFID_Read_Byte_Start_3 : BOOL := 1;
   RFID_Read_Byte_Start_4 : BOOL := 1;
   RFID_Read_Byte_Start_5 : BOOL := 1;
   RFID_Read_Byte_Start_6 : BOOL;
   RFID_Read_InProgress_1 : BOOL := 1;
   RFID_Read_InProgress_2 : BOOL;
   RFID_Read_InProgress_3 : BOOL := 1;
   RFID_Read_InProgress_4 : BOOL := 1;
   RFID_Read_InProgress_5 : BOOL := 1;
   RFID_Read_InProgress_6 : BOOL;
   RFID_Read_Start : BOOL;
   RFID_ReadData6_part_num : SINT;
   RFID_ReadData_4 : SINT;
   RFID_Write6_finshed : BOOL;
   Set_Part_Type : BOOL;
   tcoil : BOOL;
   TEST_RW : BOOL;
   TEST_RW2 : BOOL;
   Timer_RFID6_write : TIMER := (PRE := 3000);
END_VAR

ROUTINE Camera_1_Pipeline_ZZ   (* ladder *)
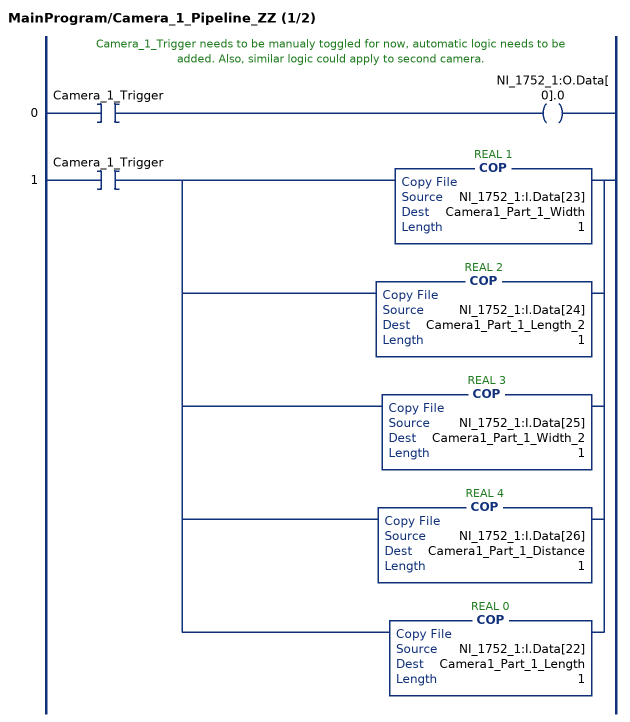
   // Camera_1_Trigger needs to be manualy toggled for now, automatic logic needs to be added. Also, similar logic could apply to second camera.
   0: XIC(Camera_1_Trigger)OTE(NI_1752_1:O.Data[0].0);
   1: XIC(Camera_1_Trigger)[COP(NI_1752_1:I.Data[23],Camera1_Part_1_Width,1) ,COP(NI_1752_1:I.Data[24],Camera1_Part_1_Length_2,1) ,COP(NI_1752_1:I.Data[25],Camera1_Part_1_Width_2,1) ,COP(NI_1752_1:I.Data[26],Camera1_Part_1_Distance,1) ,COP(NI_1752_1:I.Data[22],Camera1_Part_1_Length,1) ];
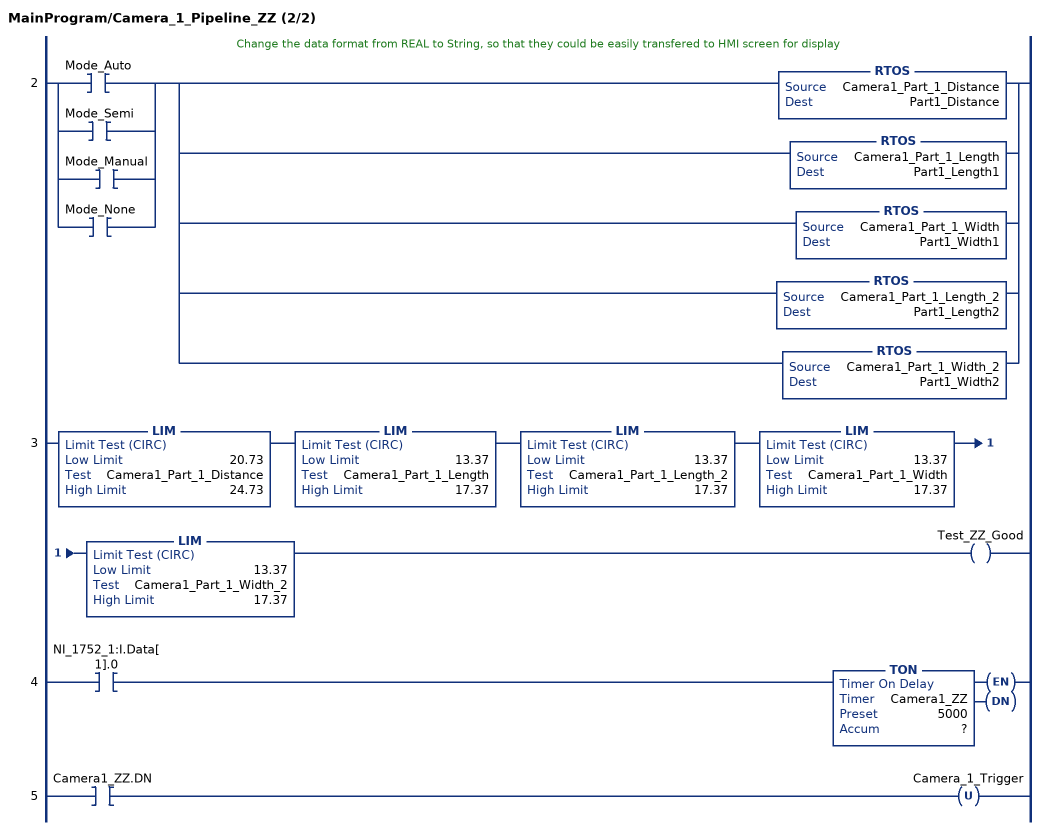
   // Change the data format from REAL to String, so that they could be easily transfered to HMI screen for display
   2: [XIC(Mode_Auto) ,XIC(Mode_Semi) ,XIC(Mode_Manual) ,XIC(Mode_None) ][RTOS(Camera1_Part_1_Distance,Part1_Distance) ,RTOS(Camera1_Part_1_Length,Part1_Length1) ,RTOS(Camera1_Part_1_Width,Part1_Width1) ,RTOS(Camera1_Part_1_Length_2,Part1_Length2) ,RTOS(Camera1_Part_1_Width_2,Part1_Width2) ];
   3: LIM(20.73,Camera1_Part_1_Distance,24.73)LIM(13.37,Camera1_Part_1_Length,17.37)LIM(13.37,Camera1_Part_1_Length_2,17.37)LIM(13.37,Camera1_Part_1_Width,17.37)LIM(13.37,Camera1_Part_1_Width_2,17.37)OTE(Test_ZZ_Good);
   4: XIC(NI_1752_1:I.Data[1].0)TON(Camera1_ZZ,?,?);
   5: XIC(Camera1_ZZ.DN)OTU(Camera_1_Trigger);
END_ROUTINE

ROUTINE Cell_1_2_VFD   (* ladder *)
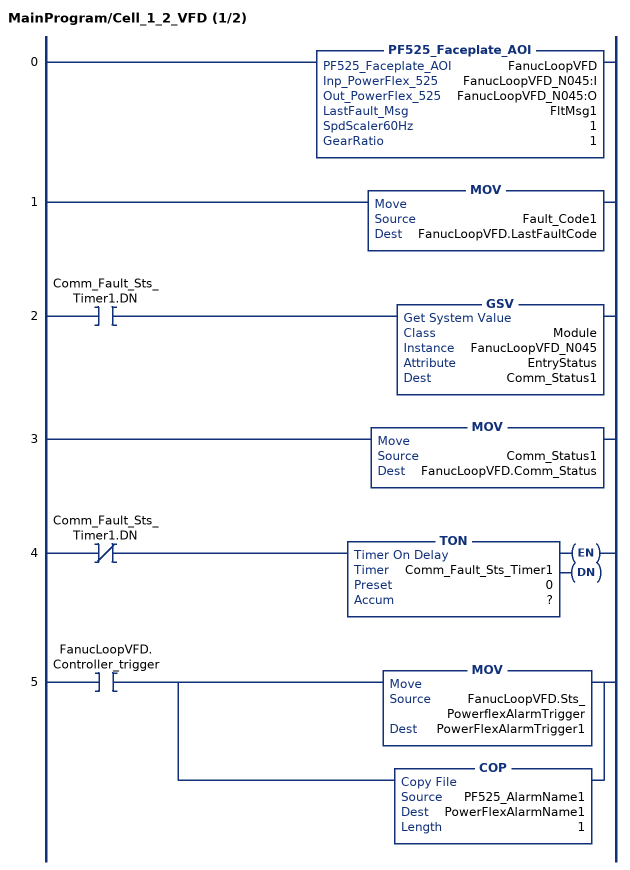
   0: PF525_Faceplate_AOI(FanucLoopVFD,FanucLoopVFD_N045:I,FanucLoopVFD_N045:O,FltMsg1,1,1);
   1: MOV(Fault_Code1,FanucLoopVFD.LastFaultCode);
   2: XIC(Comm_Fault_Sts_Timer1.DN)GSV(Module,FanucLoopVFD_N045,EntryStatus,Comm_Status1);
   3: MOV(Comm_Status1,FanucLoopVFD.Comm_Status);
   4: XIO(Comm_Fault_Sts_Timer1.DN)TON(Comm_Fault_Sts_Timer1,?,?);
   5: XIC(FanucLoopVFD.Controller_trigger)[MOV(FanucLoopVFD.Sts_PowerflexAlarmTrigger,PowerFlexAlarmTrigger1) ,COP(PF525_AlarmName1,PowerFlexAlarmName1,1) ];
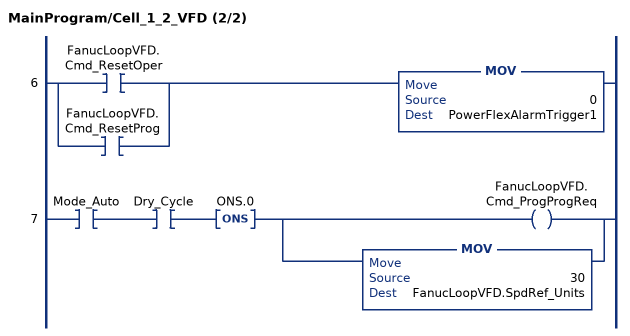
   6: [XIC(FanucLoopVFD.Cmd_ResetOper) ,XIC(FanucLoopVFD.Cmd_ResetProg) ]MOV(0,PowerFlexAlarmTrigger1);
   7: XIC(Mode_Auto)XIC(Dry_Cycle)ONS(ONS.0)[OTE(FanucLoopVFD.Cmd_ProgProgReq) ,MOV(30,FanucLoopVFD.SpdRef_Units) ];
END_ROUTINE

ROUTINE Cell_1_ZZ   (* ladder *)
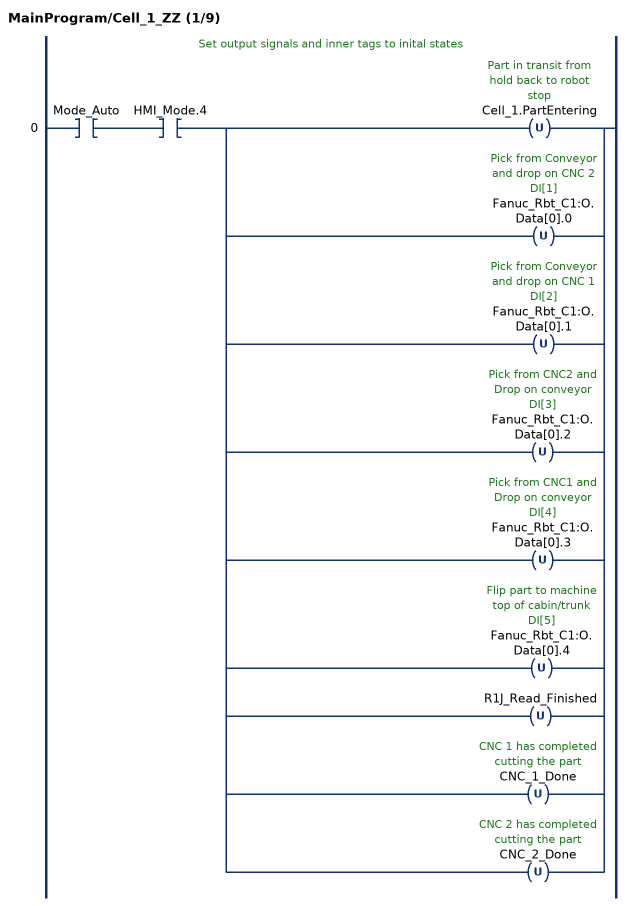
   // Set output signals and inner tags to inital states
   0: XIC(Mode_Auto)XIC(HMI_Mode.4)[OTU(Cell_1.PartEntering) ,OTU(Fanuc_Rbt_C1:O.Data[0].0) ,OTU(Fanuc_Rbt_C1:O.Data[0].1) ,OTU(Fanuc_Rbt_C1:O.Data[0].2) ,OTU(Fanuc_Rbt_C1:O.Data[0].3) ,OTU(Fanuc_Rbt_C1:O.Data[0].4) ,OTU(R1J_Read_Finished) ,OTU(CNC_1_Done) ,OTU(CNC_2_Done) ];
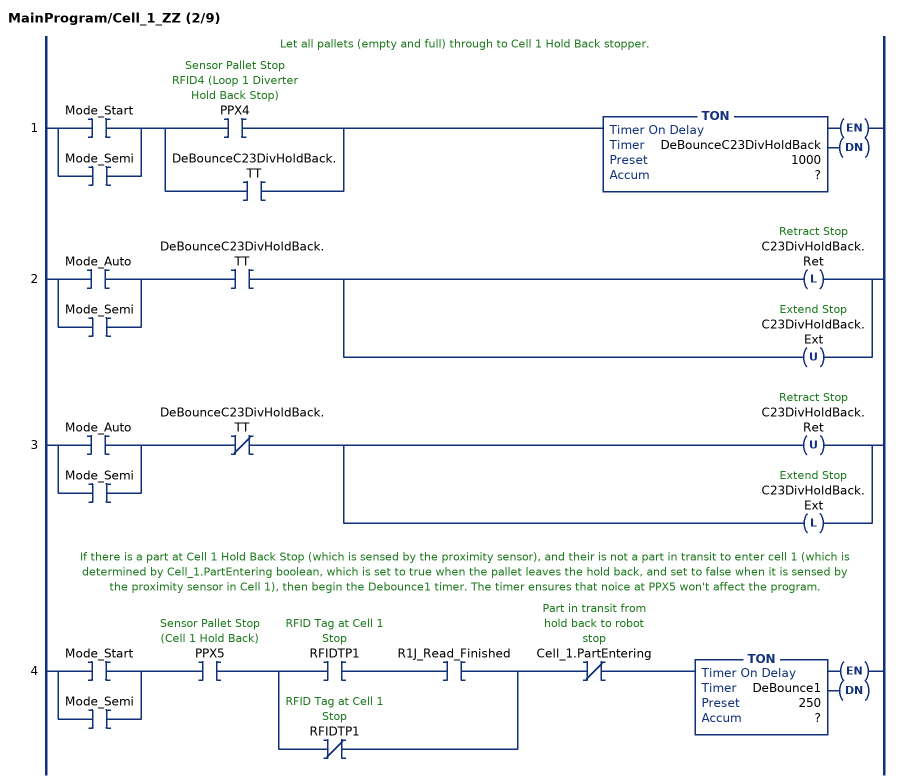
   // Let all pallets (empty and full) through to Cell 1 Hold Back stopper.
   1: [XIC(Mode_Start) ,XIC(Mode_Semi) ][XIC(PPX4) ,XIC(DeBounceC23DivHoldBack.TT) ]TON(DeBounceC23DivHoldBack,?,?);
   2: [XIC(Mode_Auto) ,XIC(Mode_Semi) ]XIC(DeBounceC23DivHoldBack.TT)[OTL(C23DivHoldBack.Ret) ,OTU(C23DivHoldBack.Ext) ];
   3: [XIC(Mode_Auto) ,XIC(Mode_Semi) ]XIO(DeBounceC23DivHoldBack.TT)[OTU(C23DivHoldBack.Ret) ,OTL(C23DivHoldBack.Ext) ];
   // If there is a part at Cell 1 Hold Back Stop (which is sensed by the proximity sensor), and their is not a part in transit to enter cell 1 (which is determined by Cell_1.PartEntering boolean, which is set to true when the pallet leaves the hold back, and set to false when it is sensed by the proximity sensor in Cell 1), then begin the Debounce1 timer. The timer ensures that noice at PPX5 won't affect the program.
   4: [XIC(Mode_Start) ,XIC(Mode_Semi) ]XIC(PPX5)[XIC(RFIDTP1) XIC(R1J_Read_Finished) ,XIO(RFIDTP1) ]XIO(Cell_1.PartEntering)TON(DeBounce1,?,?);
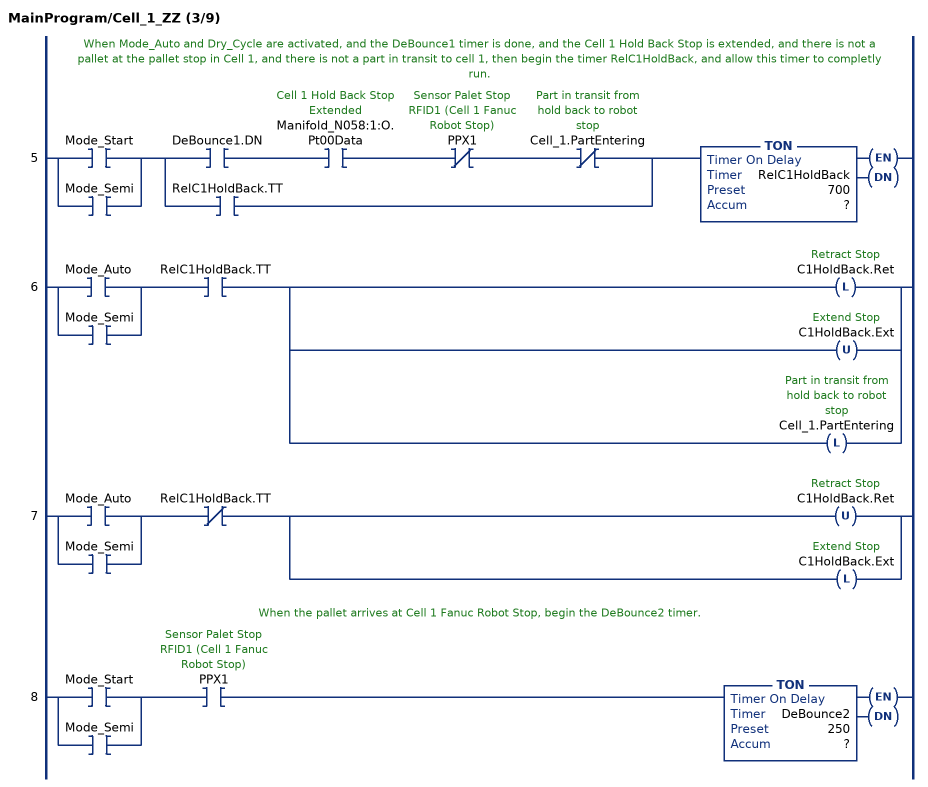
   // When Mode_Auto and Dry_Cycle are activated, and the DeBounce1 timer is done, and the Cell 1 Hold Back Stop is extended, and there is not a pallet at the pallet stop in Cell 1, and there is not a part in transit to cell 1, then begin the timer RelC1HoldBack, and allow this timer to completly run.
   5: [XIC(Mode_Start) ,XIC(Mode_Semi) ][XIC(DeBounce1.DN) XIC(Manifold_N058:1:O.Pt00Data) XIO(PPX1) XIO(Cell_1.PartEntering) ,XIC(RelC1HoldBack.TT) ]TON(RelC1HoldBack,?,?);
   6: [XIC(Mode_Auto) ,XIC(Mode_Semi) ]XIC(RelC1HoldBack.TT)[OTL(C1HoldBack.Ret) ,OTU(C1HoldBack.Ext) ,OTL(Cell_1.PartEntering) ];
   7: [XIC(Mode_Auto) ,XIC(Mode_Semi) ]XIO(RelC1HoldBack.TT)[OTU(C1HoldBack.Ret) ,OTL(C1HoldBack.Ext) ];
   // When the pallet arrives at Cell 1 Fanuc Robot Stop, begin the DeBounce2 timer.
   8: [XIC(Mode_Start) ,XIC(Mode_Semi) ]XIC(PPX1)TON(DeBounce2,?,?);
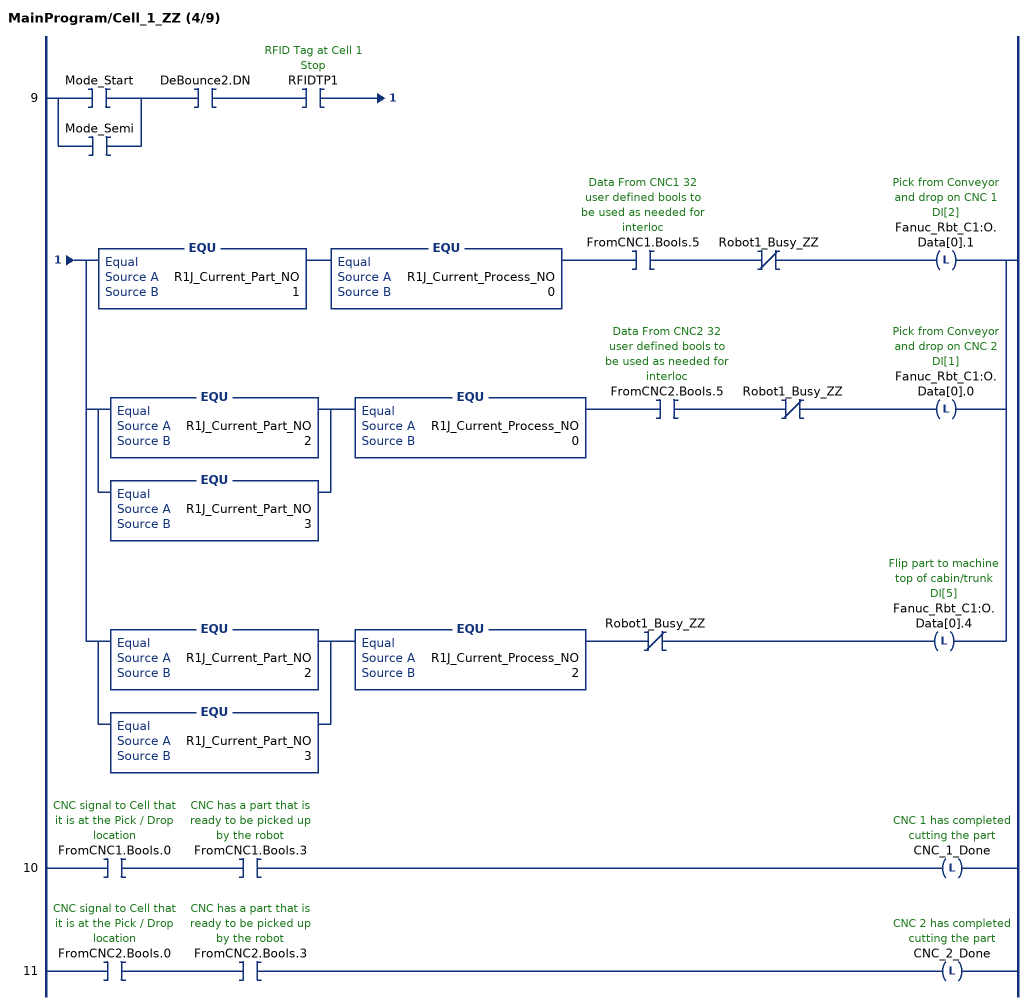
   9: [XIC(Mode_Start) ,XIC(Mode_Semi) ]XIC(DeBounce2.DN)XIC(RFIDTP1)[EQU(R1J_Current_Part_NO,1) EQU(R1J_Current_Process_NO,0) XIC(FromCNC1.Bools.5) XIO(Robot1_Busy_ZZ) OTL(Fanuc_Rbt_C1:O.Data[0].1) ,[EQU(R1J_Current_Part_NO,2) ,EQU(R1J_Current_Part_NO,3) ] EQU(R1J_Current_Process_NO,0) XIC(FromCNC2.Bools.5) XIO(Robot1_Busy_ZZ) OTL(Fanuc_Rbt_C1:O.Data[0].0) ,[EQU(R1J_Current_Part_NO,2) ,EQU(R1J_Current_Part_NO,3) ] EQU(R1J_Current_Process_NO,2) XIO(Robot1_Busy_ZZ) OTL(Fanuc_Rbt_C1:O.Data[0].4) ];
   10: XIC(FromCNC1.Bools.0)XIC(FromCNC1.Bools.3)OTL(CNC_1_Done);
   11: XIC(FromCNC2.Bools.0)XIC(FromCNC2.Bools.3)OTL(CNC_2_Done);
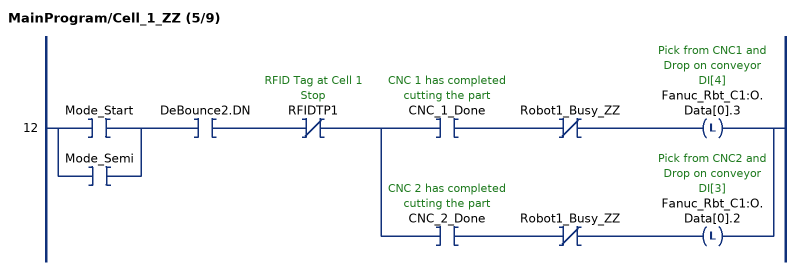
   12: [XIC(Mode_Start) ,XIC(Mode_Semi) ]XIC(DeBounce2.DN)XIO(RFIDTP1)[XIC(CNC_1_Done) XIO(Robot1_Busy_ZZ) OTL(Fanuc_Rbt_C1:O.Data[0].3) ,XIC(CNC_2_Done) XIO(Robot1_Busy_ZZ) OTL(Fanuc_Rbt_C1:O.Data[0].2) ];
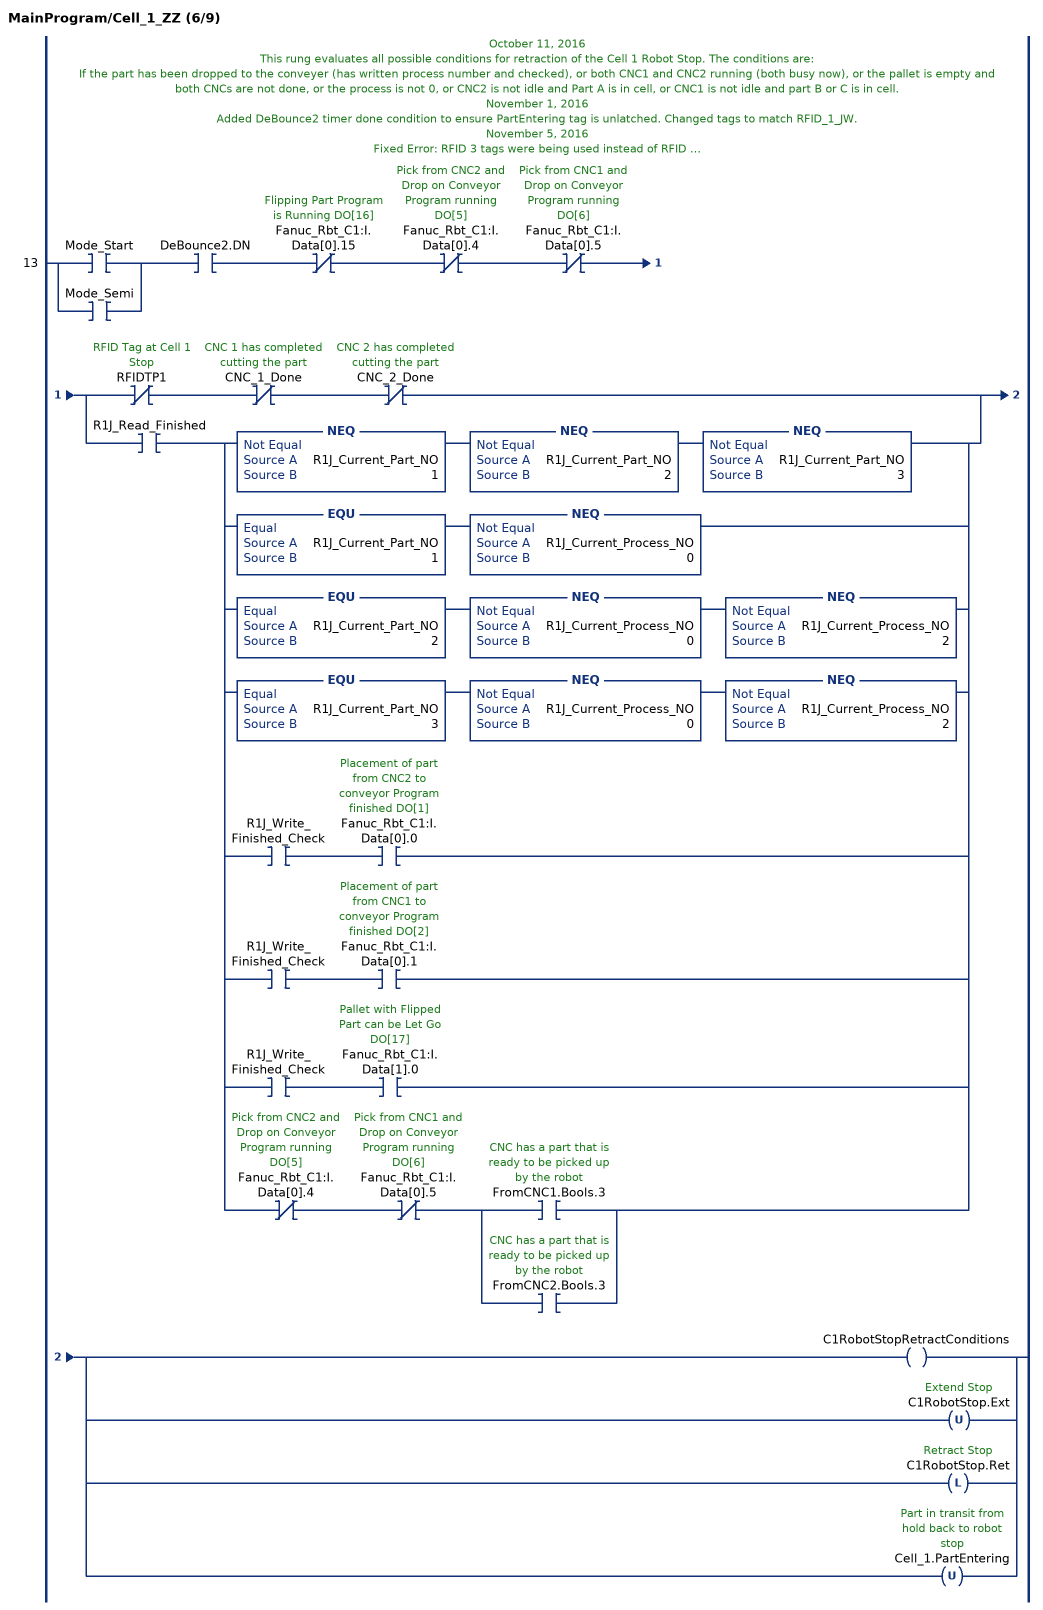
   // October 11, 2016
   // This rung evaluates all possible conditions for retraction of the Cell 1 Robot Stop. The conditions are:
   // If the part has been dropped to the conveyer (has written process number and checked), or both CNC1 and CNC2 running (both busy now), or the pallet is empty and both CNCs are not done, or the process is not 0, or CNC2 is not idle and Part A is in cell, or CNC1 is not idle and part B or C is in cell.
   // November 1, 2016
   // Added DeBounce2 timer done condition to ensure PartEntering tag is unlatched. Changed tags to match RFID_1_JW.
   // November 5, 2016
   // Fixed Error: RFID 3 tags were being used instead of RFID 1
   // November 9, 2016
   // Added Robot2_DroppedP1 and P2 FALSE conditions in front of some rungs to avoid releasing a pallet early while the robot is dropping a part from a CNC to the conveyor.
   13: [XIC(Mode_Start) ,XIC(Mode_Semi) ]XIC(DeBounce2.DN)XIO(Fanuc_Rbt_C1:I.Data[0].15)XIO(Fanuc_Rbt_C1:I.Data[0].4)XIO(Fanuc_Rbt_C1:I.Data[0].5)[XIO(RFIDTP1) XIO(CNC_1_Done) XIO(CNC_2_Done) ,XIC(R1J_Read_Finished) [[NEQ(R1J_Current_Part_NO,1) NEQ(R1J_Current_Part_NO,2) NEQ(R1J_Current_Part_NO,3) ,EQU(R1J_Current_Part_NO,1) NEQ(R1J_Current_Process_NO,0) ,EQU(R1J_Current_Part_NO,2) NEQ(R1J_Current_Process_NO,0) NEQ(R1J_Current_Process_NO,2) ,EQU(R1J_Current_Part_NO,3) NEQ(R1J_Current_Process_NO,0) NEQ(R1J_Current_Process_NO,2) ] ,XIC(R1J_Write_Finished_Check) XIC(Fanuc_Rbt_C1:I.Data[0].0) ,XIC(R1J_Write_Finished_Check) XIC(Fanuc_Rbt_C1:I.Data[0].1) ,XIC(R1J_Write_Finished_Check) XIC(Fanuc_Rbt_C1:I.Data[1].0) ,XIO(Fanuc_Rbt_C1:I.Data[0].4) XIO(Fanuc_Rbt_C1:I.Data[0].5) [XIC(FromCNC1.Bools.3) ,XIC(FromCNC2.Bools.3) ] ] ][OTE(C1RobotStopRetractConditions) ,OTU(C1RobotStop.Ext) ,OTL(C1RobotStop.Ret) ,OTU(Cell_1.PartEntering) ];
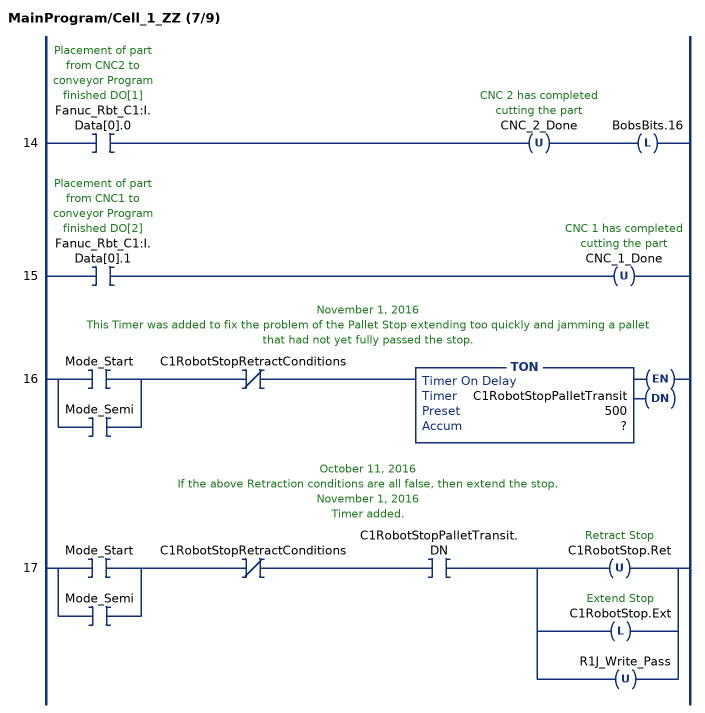
   14: XIC(Fanuc_Rbt_C1:I.Data[0].0)OTU(CNC_2_Done)OTL(BobsBits.16);
   15: XIC(Fanuc_Rbt_C1:I.Data[0].1)OTU(CNC_1_Done);
   // November 1, 2016
   // This Timer was added to fix the problem of the Pallet Stop extending too quickly and jamming a pallet that had not yet fully passed the stop.
   16: [XIC(Mode_Start) ,XIC(Mode_Semi) ]XIO(C1RobotStopRetractConditions)TON(C1RobotStopPalletTransit,?,?);
   // October 11, 2016
   // If the above Retraction conditions are all false, then extend the stop.
   // November 1, 2016
   // Timer added.
   17: [XIC(Mode_Start) ,XIC(Mode_Semi) ]XIO(C1RobotStopRetractConditions)XIC(C1RobotStopPalletTransit.DN)[OTU(C1RobotStop.Ret) ,OTL(C1RobotStop.Ext) ,OTU(R1J_Write_Pass) ];
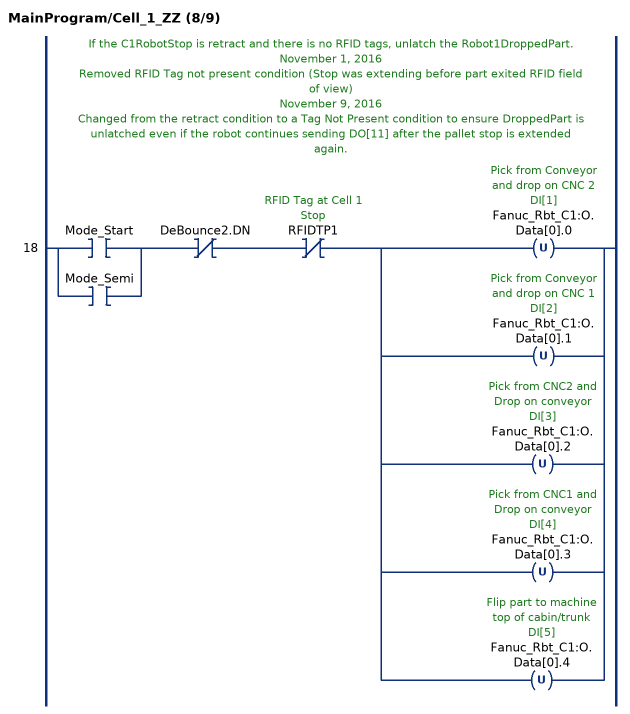
   // If the C1RobotStop is retract and there is no RFID tags, unlatch the Robot1DroppedPart.
   // November 1, 2016
   // Removed RFID Tag not present condition (Stop was extending before part exited RFID field of view)
   // November 9, 2016
   // Changed from the retract condition to a Tag Not Present condition to ensure DroppedPart is unlatched even if the robot continues sending DO[11] after the pallet stop is extended again.
   18: [XIC(Mode_Start) ,XIC(Mode_Semi) ]XIO(DeBounce2.DN)XIO(RFIDTP1)[OTU(Fanuc_Rbt_C1:O.Data[0].0) ,OTU(Fanuc_Rbt_C1:O.Data[0].1) ,OTU(Fanuc_Rbt_C1:O.Data[0].2) ,OTU(Fanuc_Rbt_C1:O.Data[0].3) ,OTU(Fanuc_Rbt_C1:O.Data[0].4) ];
